HMI_DO(Sync := HMI.HMI_DO_Index<DO_Mapping.Do_End, HMI := HMI.HMI_DO_data, Local := GVL.Dout[HMI.HMI_DO_Index], strMode => HMI.HMI_DO_data.strMode, strStatus => HMI.HMI_DO_data.strStatus);
IF HMI_DO.ENO THEN
  DO_Name:=HMI.HMI_DO_Index;
  HMI.HMI_DO_Data.strName:=Burkert.Burkert_OSCAT_BASIC.REPLACE_ALL(str:=TO_STRING(DO_Name), src:='_' , rep:=' ' );
END_IF;

HMI_8098(Sync := HMI.HMI_8098_Index<s8098_Mapping.s8098_end, HMI := HMI.HMI_8098_Data, Local := PVL.s8098[HMI.HMI_8098_Index], strNamur => HMI.HMI_8098_Data.StrNamur107);
IF HMI_8098.ENO THEN
  S8098_Name:=HMI.HMI_8098_Index;
  HMI.HMI_8098_Data.strName:=Burkert.Burkert_OSCAT_BASIC.REPLACE_ALL(str:=TO_STRING(s8098_Name), src:='_' , rep:=' ' );
END_IF;

_Burkert_HMI_ME44AI_Sync187_OUT := Burkert.HMI_ME44AI_Sync(EN := HMI.HMI_ME44AI_Index<ME44AI_Mapping.ME44_AI_End, Local := Network.ME44_AI[HMI.HMI_ME44AI_Index], HMI := HMI.HMI_ME44AI_data, ENO => _Burkert_HMI_ME44AI_Sync187_ENO);
IF _Burkert_HMI_ME44AI_Sync187_ENO THEN
  ME44AI_Name:=HMI.HMI_ME44AI_Index;
  HMI.HMI_ME44AI_Data.strName:=Burkert.Burkert_OSCAT_BASIC.REPLACE_ALL(str:=TO_STRING(ME44AI_Name), src:='_' , rep:=' ' );
END_IF;
END_PROGRAM

PROGRAM VFD_Manager
  VAR
    VFD_101A_CTRL : Burkert.Eaton_DM1;
    VFD_101B_CTRL : Burkert.Eaton_DM1;
    VFD_102A_CTRL : Burkert.Eaton_DM1;
    VFD_102B_CTRL : Burkert.Eaton_DM1;
    VFD_102C_CTRL : Burkert.Eaton_DM1;
    VFD_102D_CTRL : Burkert.Eaton_DM1;
    VFD_102E_CTRL : Burkert.Eaton_DM1;
    VFD_102F_CTRL : Burkert.Eaton_DM1;
    VFD_102G_CTRL : Burkert.Eaton_DM1;
    VFD_102H_CTRL : Burkert.Eaton_DM1;
    VFD_201_CTRL : Burkert.Eaton_DM1;
    VFD_201B_CTRL : Burkert.Eaton_DM1;
    VFD_202_CTRL : Burkert.Eaton_DM1;
    VFD_202B_CTRL : Burkert.Eaton_DM1;
    VFD_203_CTRL : Burkert.Eaton_DM1;
  END_VAR

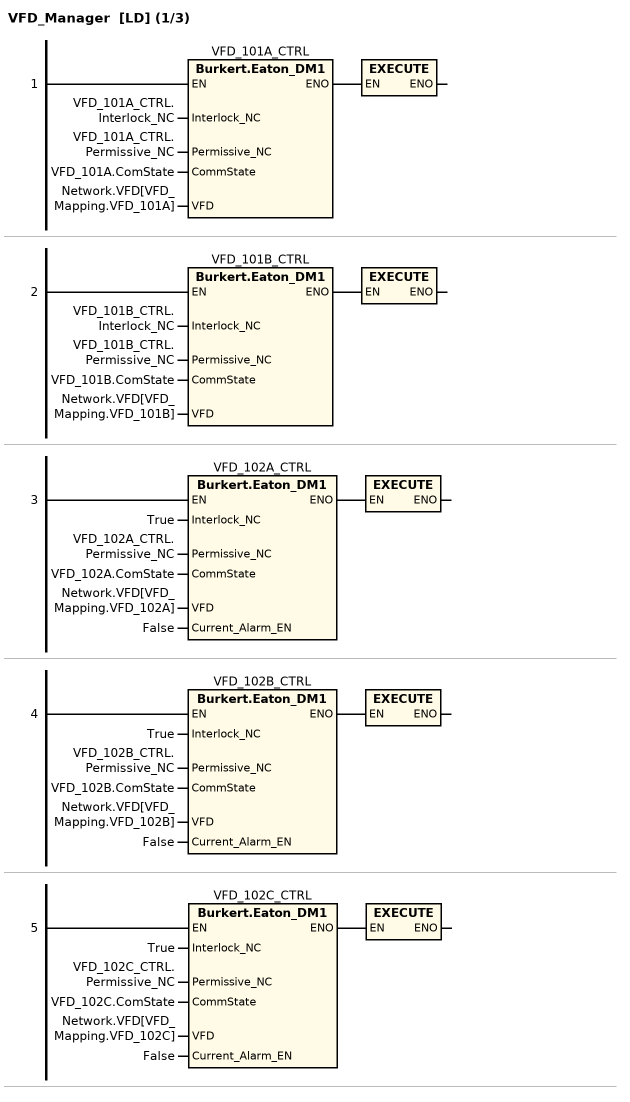
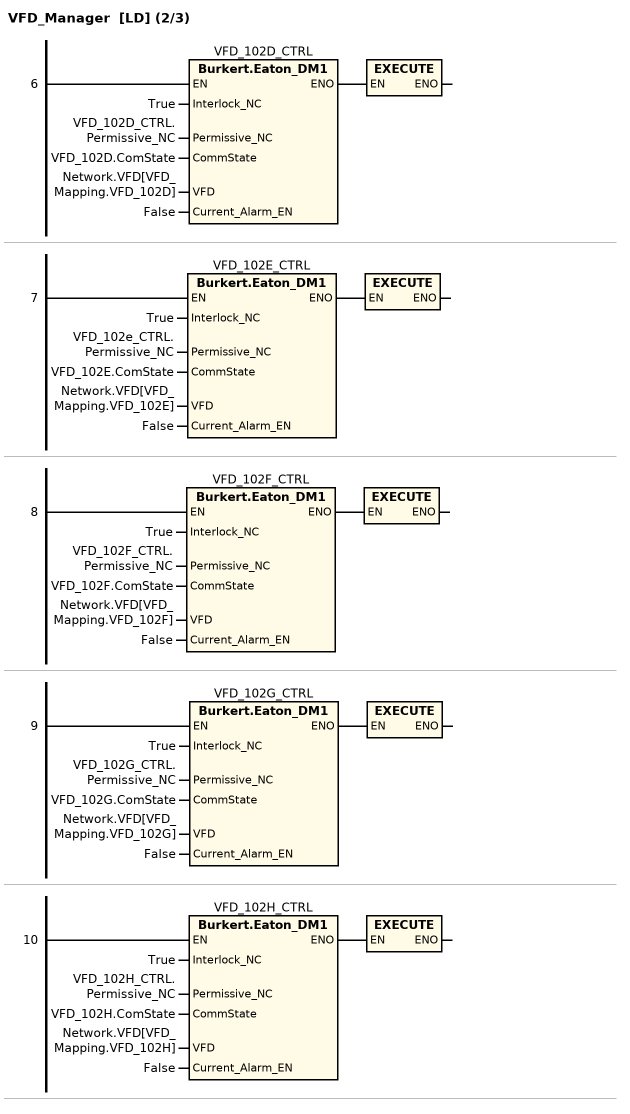
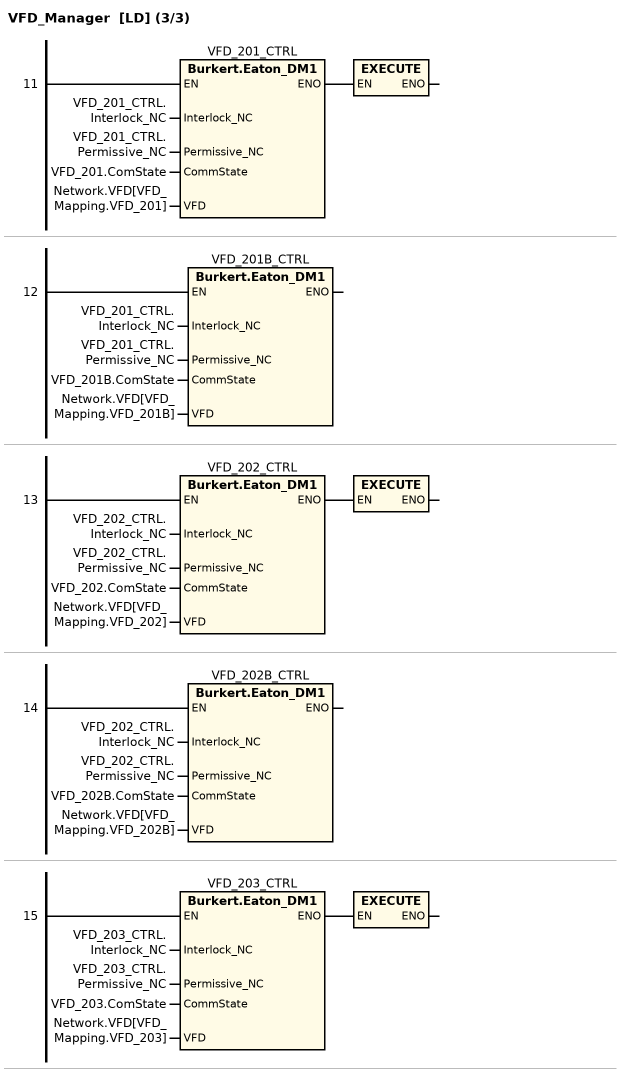
(* LD diagram, written out as Structured Text *)

VFD_101A_CTRL(Interlock_NC := VFD_101A_CTRL.Interlock_NC, Permissive_NC := VFD_101A_CTRL.Permissive_NC, CommState := VFD_101A.ComState, VFD := Network.VFD[VFD_Mapping.VFD_101A]);
IF VFD_101A_CTRL.ENO THEN
  VFD_101A_CTRL.Permissive_NC:= (GVL.s3363[s3363_mapping.ACV_101].Valve_Actual>5
  	) AND (
  	GVL.LS[LS_Mapping.LSLL_101].Status.eStatus=Burkert.DI_Status.Liquid_Detected AND
  	GVL.LS[Ls_mapping.LSHH_201].Status.eStatus=Burkert.DI_Status.No_Liquid_Detected);
  
  
  VFD_101A_CTRL.Interlock_NC:=TRUE;//(
  	//GVL.LS[LS_Mapping.LSLL_101].Status.eStatus=Burkert.DI_Status.Liquid_Detected AND
  	//GVL.LS[Ls_mapping.LSHH_201].Status.eStatus=Burkert.DI_Status.No_Liquid_Detected);
END_IF;

VFD_101B_CTRL(Interlock_NC := VFD_101B_CTRL.Interlock_NC, Permissive_NC := VFD_101B_CTRL.Permissive_NC, CommState := VFD_101B.ComState, VFD := Network.VFD[VFD_Mapping.VFD_101B]);
IF VFD_101B_CTRL.ENO THEN
  VFD_101B_CTRL.Permissive_NC:=(GVL.s3363[s3363_mapping.ACV_102].Valve_Actual>5 ) AND 
  	(GVL.LS[LS_Mapping.LSLL_101].Status.eStatus=Burkert.DI_Status.Liquid_Detected AND
  	GVL.LS[Ls_mapping.LSHH_201].Status.eStatus=Burkert.DI_Status.No_Liquid_Detected) ;
  	
  	VFD_101B_CTRL.Interlock_NC:=TRUE;//
  //(GVL.LS[LS_Mapping.LSLL_101].Status.eStatus=Burkert.DI_Status.Liquid_Detected AND GVL.LS[Ls_mapping.LSHH_201].Status.eStatus=Burkert.DI_Status.No_Liquid_Detected);
END_IF;

VFD_102A_CTRL(Interlock_NC := True, Permissive_NC := VFD_102A_CTRL.Permissive_NC, CommState := VFD_102A.ComState, VFD := Network.VFD[VFD_Mapping.VFD_102A], Current_Alarm_EN := False);
IF VFD_102A_CTRL.ENO THEN
  VFD_102A_CTRL.Permissive_NC:=(
  	NOT(PVL.AIT[AIT_Mapping.LT_101_P].Status.eStatus=Burkert.eSensor_Status.Low_Low_Alarm)
  	);
END_IF;

VFD_102B_CTRL(Interlock_NC := True, Permissive_NC := VFD_102B_CTRL.Permissive_NC, CommState := VFD_102B.ComState, VFD := Network.VFD[VFD_Mapping.VFD_102B], Current_Alarm_EN := False);
IF VFD_102B_CTRL.ENO THEN
  VFD_102B_CTRL.Permissive_NC:=(
  	NOT(PVL.AIT[AIT_Mapping.LT_101_P].Status.eStatus=Burkert.eSensor_Status.Low_Low_Alarm)
  	);
END_IF;

VFD_102C_CTRL(Interlock_NC := True, Permissive_NC := VFD_102C_CTRL.Permissive_NC, CommState := VFD_102C.ComState, VFD := Network.VFD[VFD_Mapping.VFD_102C], Current_Alarm_EN := False);
IF VFD_102C_CTRL.ENO THEN
  VFD_102C_CTRL.Permissive_NC:=(
  	NOT(PVL.AIT[AIT_Mapping.LT_101_P].Status.eStatus=Burkert.eSensor_Status.Low_Low_Alarm)
  	);
END_IF;

VFD_102D_CTRL(Interlock_NC := True, Permissive_NC := VFD_102D_CTRL.Permissive_NC, CommState := VFD_102D.ComState, VFD := Network.VFD[VFD_Mapping.VFD_102D], Current_Alarm_EN := False);
IF VFD_102D_CTRL.ENO THEN
  VFD_102D_CTRL.Permissive_NC:=(
  	NOT(PVL.AIT[AIT_Mapping.LT_101_P].Status.eStatus=Burkert.eSensor_Status.Low_Low_Alarm)
  	);
END_IF;

VFD_102E_CTRL(Interlock_NC := True, Permissive_NC := VFD_102e_CTRL.Permissive_NC, CommState := VFD_102E.ComState, VFD := Network.VFD[VFD_Mapping.VFD_102E], Current_Alarm_EN := False);
IF VFD_102E_CTRL.ENO THEN
  VFD_102E_CTRL.Permissive_NC:=(
  	NOT(PVL.AIT[AIT_Mapping.LT_201].Status.eStatus=Burkert.eSensor_Status.Low_Low_Alarm)
  	);
END_IF;

VFD_102F_CTRL(Interlock_NC := True, Permissive_NC := VFD_102F_CTRL.Permissive_NC, CommState := VFD_102F.ComState, VFD := Network.VFD[VFD_Mapping.VFD_102F], Current_Alarm_EN := False);
IF VFD_102F_CTRL.ENO THEN
  VFD_102F_CTRL.Permissive_NC:=(
  	NOT(PVL.AIT[AIT_Mapping.LT_201].Status.eStatus=Burkert.eSensor_Status.Low_Low_Alarm)
  	);
END_IF;

VFD_102G_CTRL(Interlock_NC := True, Permissive_NC := VFD_102G_CTRL.Permissive_NC, CommState := VFD_102G.ComState, VFD := Network.VFD[VFD_Mapping.VFD_102G], Current_Alarm_EN := False);
IF VFD_102G_CTRL.ENO THEN
  VFD_102G_CTRL.Permissive_NC:=(
  	NOT(PVL.AIT[AIT_Mapping.LT_201].Status.eStatus=Burkert.eSensor_Status.Low_Low_Alarm)
  	);
END_IF;

VFD_102H_CTRL(Interlock_NC := True, Permissive_NC := VFD_102H_CTRL.Permissive_NC, CommState := VFD_102H.ComState, VFD := Network.VFD[VFD_Mapping.VFD_102H], Current_Alarm_EN := False);
IF VFD_102H_CTRL.ENO THEN
  VFD_102H_CTRL.Permissive_NC:=(
  	NOT(PVL.AIT[AIT_Mapping.LT_201].Status.eStatus=Burkert.eSensor_Status.Low_Low_Alarm)
  	);
END_IF;

VFD_201_CTRL(Interlock_NC := VFD_201_CTRL.Interlock_NC, Permissive_NC := VFD_201_CTRL.Permissive_NC, CommState := VFD_201.ComState, VFD := Network.VFD[VFD_Mapping.VFD_201]);
IF VFD_201_CTRL.ENO THEN
  VFD_201_CTRL.Permissive_NC:=(GVL.s3363[s3363_mapping.ACV_201].Valve_Actual>10) AND 
  	(
  	(GVL.LS[LS_Mapping.LSHH_204].Status.eStatus=Burkert.DI_Status.No_Liquid_Detected OR GVL.LS[LS_Mapping.LSHH_204].Status.eStatus=Burkert.DI_Status.No_Liquid_Detected_Alarm) AND (GVL.LS[LS_mapping.LSLL_202].Status.eStatus=Burkert.DI_Status.Liquid_Detected)
  	);
  
  VFD_201_CTRL.Interlock_NC:=TRUE;//
  //((GVL.LS[LS_Mapping.LSHH_204].Status.eStatus=Burkert.DI_Status.No_Liquid_Detected OR GVL.LS[LS_Mapping.LSHH_204].Status.eStatus=Burkert.DI_Status.No_Liquid_Detected_Alarm) AND (GVL.LS[LS_mapping.LSLL_202].Status.eStatus=Burkert.DI_Status.Liquid_Detected));
END_IF;

VFD_201B_CTRL(Interlock_NC := VFD_201_CTRL.Interlock_NC, Permissive_NC := VFD_201_CTRL.Permissive_NC, CommState := VFD_201B.ComState, VFD := Network.VFD[VFD_Mapping.VFD_201B]);

VFD_202_CTRL(Interlock_NC := VFD_202_CTRL.Interlock_NC, Permissive_NC := VFD_202_CTRL.Permissive_NC, CommState := VFD_202.ComState, VFD := Network.VFD[VFD_Mapping.VFD_202]);
IF VFD_202_CTRL.ENO THEN
  VFD_202_CTRL.Permissive_NC:=(
  	(GVL.LS[LS_Mapping.LSLL_205].Status.eStatus=Burkert.DI_Status.Liquid_Detected) AND
  		(GVL.Filter_Path_Available OR 
  		(GVL.s3363[s3363_Mapping.ACV_203].Valve_Actual>5 AND GVL.s3363[s3363_Mapping.ACV_206].Valve_Actual>5)
  			)
  	);
  (*		
  		(GVL.s3363[s3363_Mapping.ACV_203].Valve_Actual>5 AND GVL.s3363[s3363_Mapping.ACV_206].Valve_Actual>5) OR
  		(	GVL.s3363[s3363_Mapping.ACV_207].Valve_Actual>5 OR
  			GVL.s3363[s3363_Mapping.ACV_208].Valve_Actual>5 OR
  			GVL.s3363[s3363_Mapping.ACV_213].Valve_Actual>5 OR
  			GVL.s3363[s3363_Mapping.ACV_214].Valve_Actual>5 OR
  			GVL.s3363[s3363_Mapping.ACV_219].Valve_Actual>5)
  	) AND	(
  		GVL.s3363[s3363_Mapping.ACV_224].Valve_Actual>5 OR
  		GVL.s3363[s3363_Mapping.ACV_225].Valve_Actual>5 OR
  		GVL.s3363[s3363_Mapping.ACV_226].Valve_Actual>5)	
  )	OR
  PVL.Z202_Config.Task.eTask=eZ202_Task.Drain_P202;
  *)
  
  
  
  VFD_202_CTRL.Interlock_NC:=TRUE;//(GVL.LS[LS_Mapping.LSLL_203].Status.eStatus=Burkert.DI_Status.Liquid_Detected);
END_IF;

VFD_202B_CTRL(Interlock_NC := VFD_202_CTRL.Interlock_NC, Permissive_NC := VFD_202_CTRL.Permissive_NC, CommState := VFD_202B.ComState, VFD := Network.VFD[VFD_Mapping.VFD_202B]);

VFD_203_CTRL(Interlock_NC := VFD_203_CTRL.Interlock_NC, Permissive_NC := VFD_203_CTRL.Permissive_NC, CommState := VFD_203.ComState, VFD := Network.VFD[VFD_Mapping.VFD_203]);
IF VFD_203_CTRL.ENO THEN
  VFD_203_CTRL.Permissive_NC:=(
  	(GVL.LS[LS_Mapping.LSLL_203].Status.eStatus=Burkert.DI_Status.Liquid_Detected) AND 
  	(GVL.s3363[s3363_Mapping.ACV_203].Valve_Actual>5 OR
  	(GVL.s3363[s3363_Mapping.ACV_206].Valve_Actual>6 AND GVL.Filter_Path_Available)
  	));// OR
  	//PVL.Z202_Config.Task.eTask=eZ202_Task.Drain_P203;
  	
  VFD_203_CTRL.Interlock_NC:=True;//(GVL.LS[LS_Mapping.LSLL_203].Status.eStatus=Burkert.DI_Status.Liquid_Detected);
END_IF;
END_PROGRAM

PROGRAM Stride_IO
  VAR
    Z201_RTD_Manager : Burkert.MB0_RTD;
    Z202_DO_Manager : Burkert.SIO_MB12CDR;
    tFIT : Burkert.cBase_FIT;
    tSensor : Burkert.cAnalog_Sensor;
  END_VAR

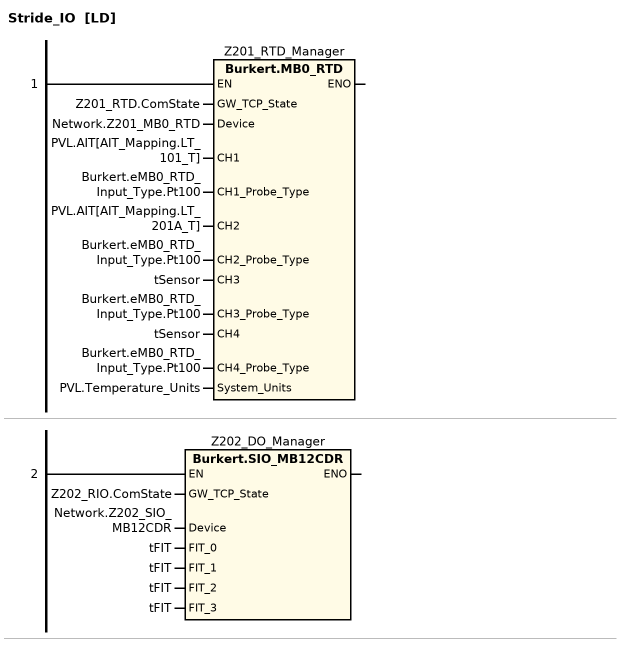
(* LD diagram, written out as Structured Text *)

Z201_RTD_Manager(GW_TCP_State := Z201_RTD.ComState, Device := Network.Z201_MB0_RTD, CH1 := PVL.AIT[AIT_Mapping.LT_101_T], CH1_Probe_Type := Burkert.eMB0_RTD_Input_Type.Pt100, CH2 := PVL.AIT[AIT_Mapping.LT_201A_T], CH2_Probe_Type := Burkert.eMB0_RTD_Input_Type.Pt100, CH3 := tSensor, CH3_Probe_Type := Burkert.eMB0_RTD_Input_Type.Pt100, CH4 := tSensor, CH4_Probe_Type := Burkert.eMB0_RTD_Input_Type.Pt100, System_Units := PVL.Temperature_Units);

Z202_DO_Manager(GW_TCP_State := Z202_RIO.ComState, Device := Network.Z202_SIO_MB12CDR, FIT_0 := tFIT, FIT_1 := tFIT, FIT_2 := tFIT, FIT_3 := tFIT);
END_PROGRAM

PROGRAM RCP_Manager
  VAR
    RecipeManCommands : RecipeManCommands;
    Save_Response : DWORD;
    Load_Response : DWORD;
    Storage_Response : BOOL;
    Load_Ton : ton;
    Save_Ton : Ton;
    Auto_Load_Ton : Ton;
    File_Save : BOOL;
    File_Save_Response : DWORD;
    R_Trig_0 : R_Trig;
    Save_R_trig : R_trig;
  END_VAR

            RecipeManCommands();
Storage_Response:=RecipeManCommands.SetStoragePath('RCP/');
//RecipeManCommands.GetRecipeNames(RecipeDefinitionName:='PersistentVariables',pStrings:=ADR(RCP_Names),iSize:=10,iStartIndex:=0);
Save_R_trig(CLK:=GVL.RCP_Save);
IF Save_R_trig.Q THEN 
	Save_Response:=16#FFFF; 
	PVL.RCP_Count:=PVL.RCP_Count+1;
END_IF;


IF GVL.RCP_Save THEN 
	//Save_Response:=16#FFFF;	
	Save_Response:=ReadAndSave();
	END_IF;
IF GVL.RCP_Load THEN	Load_Response:=LoadAndWrite(); END_IF;


Save_ton(In:=GVL.RCP_Save AND NOT(Save_Response=16#FFFF),PT:=T#2S);
IF Save_Ton.Q THEN GVL.RCP_Save:=FALSE; END_IF;




Load_ton(In:=GVL.RCP_Load,PT:=T#2S);
IF Load_Ton.Q THEN		
	GVL.RCP_Load :=FALSE;
	PVl.RCP_Loaded:=TRUE;
	END_IF;

Auto_Load_Ton(IN:=NOT(PVl.RCP_Loaded),PT:=T#10S);

IF Auto_load_Ton.Q THEN GVL.RCP_Load:=TRUE;	END_IF;
//IF GVL.Day_Seconds=30500 THEN GVL.RCP_Save:=TRUE; END_IF;
R_Trig_0(CLK:=GVL.RCP_Save);



//IF File_Save THEN 
//	File_Save_Response:=RecipeManCommands.SaveRecipe	(RecipeDefinitionName:='PersistentVariables',RecipeName:='Day_27');//,FileName:='BackUp_1.txtrecipe'); 
///END_IF;
          

METHOD ReadAndSave : DWORD
                  //ReadAndSave:=RecipeManCommands.ReadAndSaveRecipe(RecipeDefinitionName:='Vars',RecipeName:='BackUp');
//ReadAndSave:=RecipeManCommands.ReadRecipe	(RecipeDefinitionName:='PersistentVariables',RecipeName:='BackUp');
RecipeManCommands.CreateRecipe(RecipeDefinitionName:='Vars',RecipeName:='BackUp');
ReadAndSave:=RecipeManCommands.ReadAndSaveRecipeAs	(RecipeDefinitionName:='Vars',RecipeName:='BackUp',FileName:='BackUp.Vars.txtrecipe');

                
END_METHOD

METHOD LoadAndWrite : DWORD
                  //LoadAndWrite:=RecipeManCommands.LoadAndWriteRecipe(RecipeDefinitionName:='Recipes',RecipeName:='BackUp');

LoadAndWrite:=RecipeManCommands.LoadFromAndWriteRecipe(FileName:='BackUp.Vars.txtrecipe',RecipeDefinitionName:='Vars',RecipeName:='BackUp');
                
END_METHOD
END_PROGRAM

PROGRAM LS_Manager
  VAR
    LSHH_201_CTRL : Burkert.LS_UDFB;
    LSLL_202_CTRL : Burkert.LS_UDFB;
    LSLL_101_CTRL : Burkert.LS_UDFB;
    LSHH_206_CTRL : Burkert.LS_UDFB;
    LSLL_210_CTRL : Burkert.LS_UDFB;
    LSHH_208_CTRL : Burkert.LS_UDFB;
    LSLL_212_CTRL : Burkert.LS_UDFB;
    LSHH_209_CTRL : Burkert.LS_UDFB;
    LSLL_213_CTRL : Burkert.LS_UDFB;
    LSHH_207_CTRL : Burkert.LS_UDFB;
    LSLL_211_CTRL : Burkert.LS_UDFB;
    LSHH_204_CTRL : Burkert.LS_UDFB;
    LSLL_205_CTRL : Burkert.LS_UDFB;
    LSLL_203_CTRL : Burkert.LS_UDFB;
  END_VAR

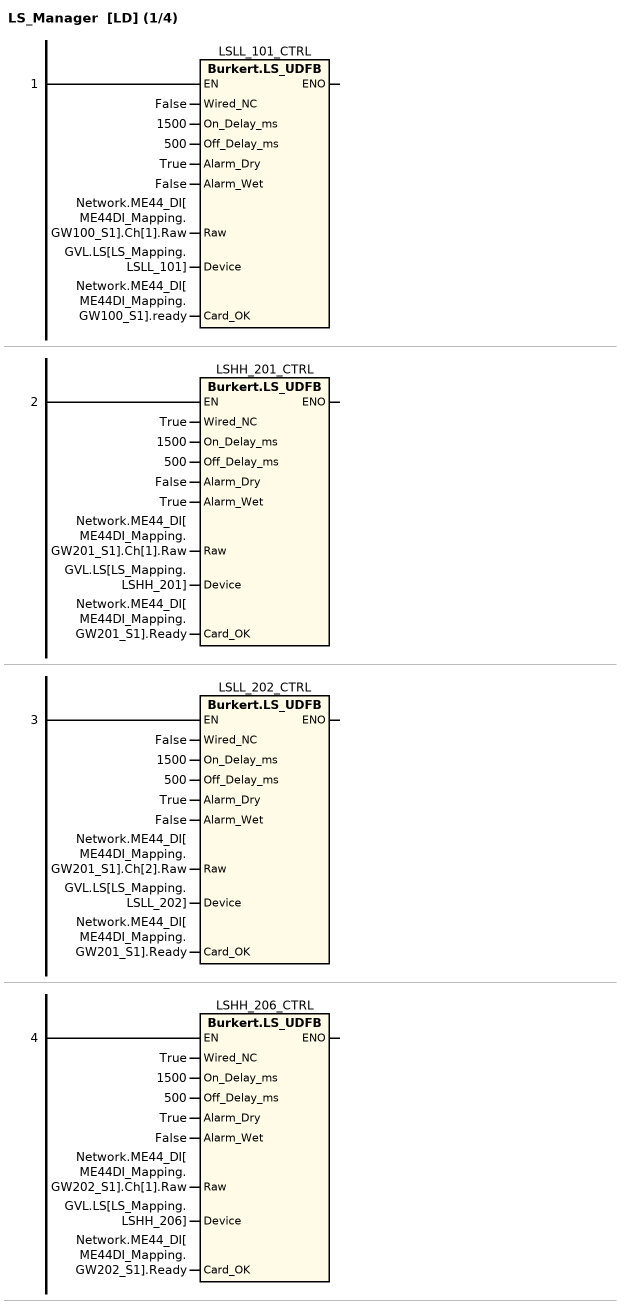
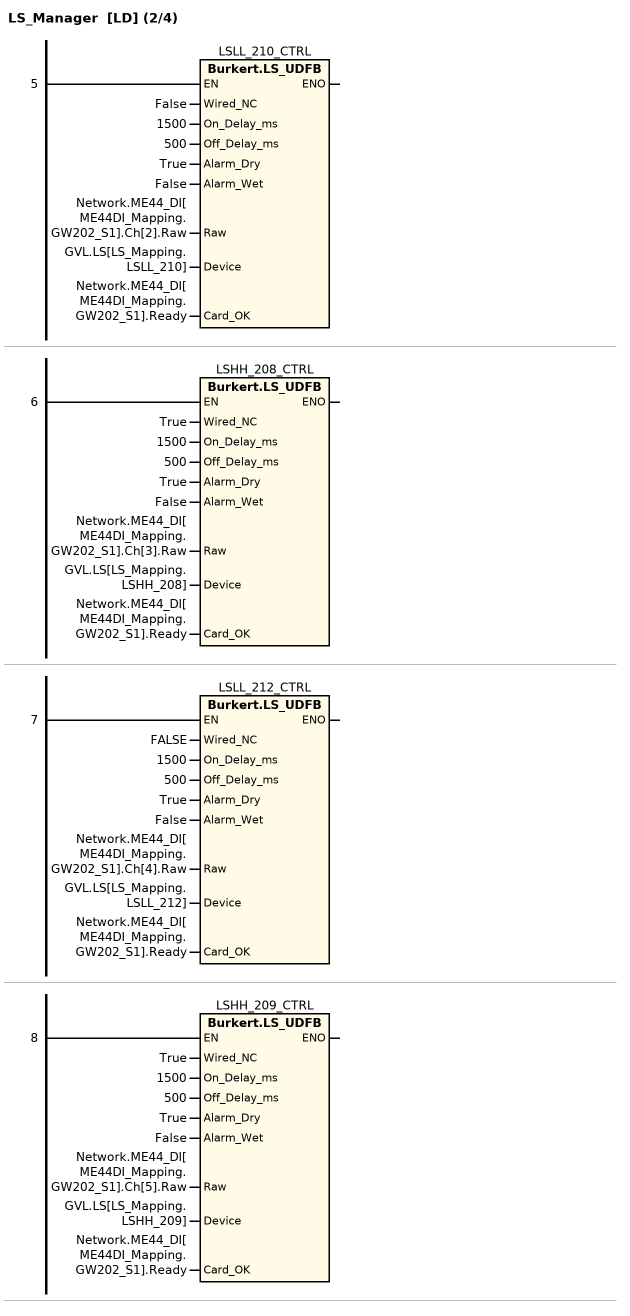
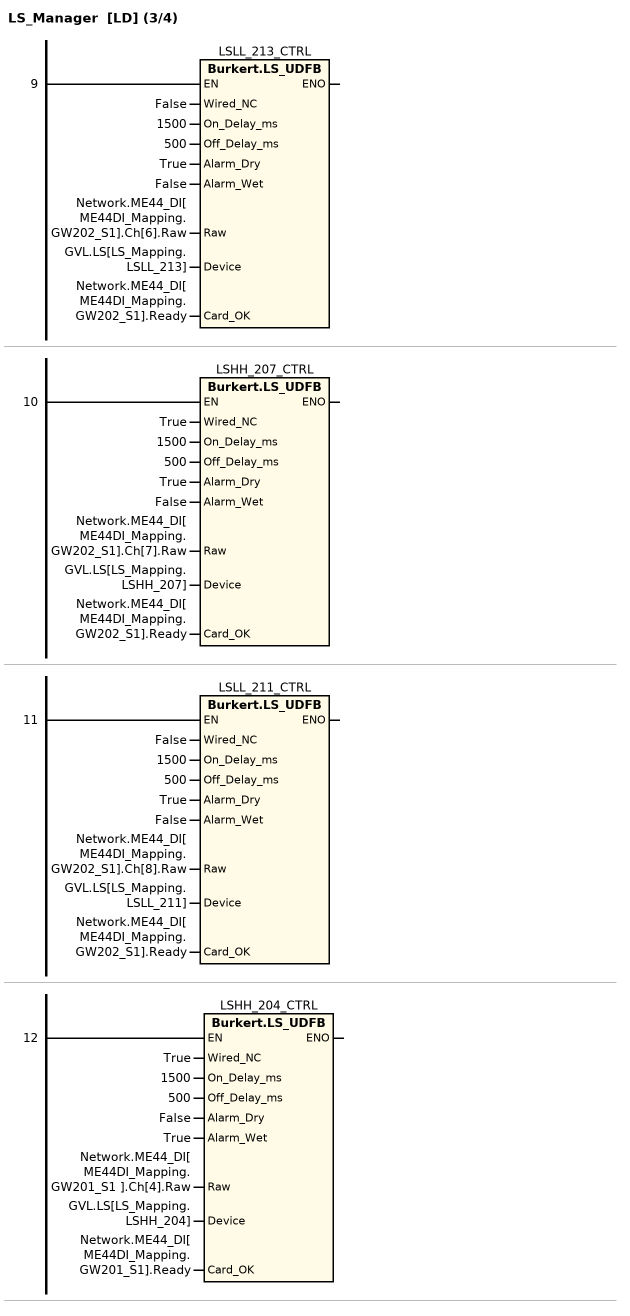
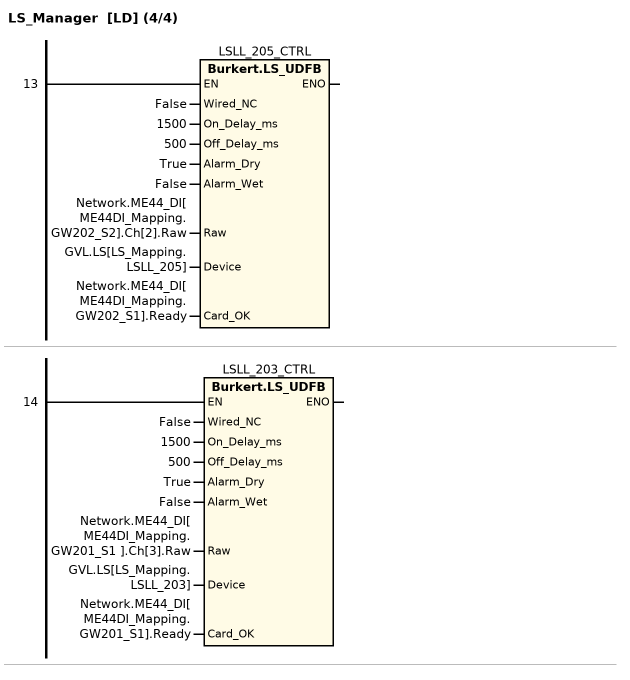
(* LD diagram, written out as Structured Text *)

LSLL_101_CTRL(Wired_NC := False, On_Delay_ms := 1500, Off_Delay_ms := 500, Alarm_Dry := True, Alarm_Wet := False, Raw := Network.ME44_DI[ME44DI_Mapping.GW100_S1].Ch[1].Raw, Device := GVL.LS[LS_Mapping.LSLL_101], Card_OK := Network.ME44_DI[ME44DI_Mapping.GW100_S1].ready);

LSHH_201_CTRL(Wired_NC := True, On_Delay_ms := 1500, Off_Delay_ms := 500, Alarm_Dry := False, Alarm_Wet := True, Raw := Network.ME44_DI[ME44DI_Mapping.GW201_S1].Ch[1].Raw, Device := GVL.LS[LS_Mapping.LSHH_201], Card_OK := Network.ME44_DI[ME44DI_Mapping.GW201_S1].Ready);

LSLL_202_CTRL(Wired_NC := False, On_Delay_ms := 1500, Off_Delay_ms := 500, Alarm_Dry := True, Alarm_Wet := False, Raw := Network.ME44_DI[ME44DI_Mapping.GW201_S1].Ch[2].Raw, Device := GVL.LS[LS_Mapping.LSLL_202], Card_OK := Network.ME44_DI[ME44DI_Mapping.GW201_S1].Ready);

LSHH_206_CTRL(Wired_NC := True, On_Delay_ms := 1500, Off_Delay_ms := 500, Alarm_Dry := True, Alarm_Wet := False, Raw := Network.ME44_DI[ME44DI_Mapping.GW202_S1].Ch[1].Raw, Device := GVL.LS[LS_Mapping.LSHH_206], Card_OK := Network.ME44_DI[ME44DI_Mapping.GW202_S1].Ready);

LSLL_210_CTRL(Wired_NC := False, On_Delay_ms := 1500, Off_Delay_ms := 500, Alarm_Dry := True, Alarm_Wet := False, Raw := Network.ME44_DI[ME44DI_Mapping.GW202_S1].Ch[2].Raw, Device := GVL.LS[LS_Mapping.LSLL_210], Card_OK := Network.ME44_DI[ME44DI_Mapping.GW202_S1].Ready);

LSHH_208_CTRL(Wired_NC := True, On_Delay_ms := 1500, Off_Delay_ms := 500, Alarm_Dry := True, Alarm_Wet := False, Raw := Network.ME44_DI[ME44DI_Mapping.GW202_S1].Ch[3].Raw, Device := GVL.LS[LS_Mapping.LSHH_208], Card_OK := Network.ME44_DI[ME44DI_Mapping.GW202_S1].Ready);

LSLL_212_CTRL(Wired_NC := FALSE, On_Delay_ms := 1500, Off_Delay_ms := 500, Alarm_Dry := True, Alarm_Wet := False, Raw := Network.ME44_DI[ME44DI_Mapping.GW202_S1].Ch[4].Raw, Device := GVL.LS[LS_Mapping.LSLL_212], Card_OK := Network.ME44_DI[ME44DI_Mapping.GW202_S1].Ready);

LSHH_209_CTRL(Wired_NC := True, On_Delay_ms := 1500, Off_Delay_ms := 500, Alarm_Dry := True, Alarm_Wet := False, Raw := Network.ME44_DI[ME44DI_Mapping.GW202_S1].Ch[5].Raw, Device := GVL.LS[LS_Mapping.LSHH_209], Card_OK := Network.ME44_DI[ME44DI_Mapping.GW202_S1].Ready);

LSLL_213_CTRL(Wired_NC := False, On_Delay_ms := 1500, Off_Delay_ms := 500, Alarm_Dry := True, Alarm_Wet := False, Raw := Network.ME44_DI[ME44DI_Mapping.GW202_S1].Ch[6].Raw, Device := GVL.LS[LS_Mapping.LSLL_213], Card_OK := Network.ME44_DI[ME44DI_Mapping.GW202_S1].Ready);

LSHH_207_CTRL(Wired_NC := True, On_Delay_ms := 1500, Off_Delay_ms := 500, Alarm_Dry := True, Alarm_Wet := False, Raw := Network.ME44_DI[ME44DI_Mapping.GW202_S1].Ch[7].Raw, Device := GVL.LS[LS_Mapping.LSHH_207], Card_OK := Network.ME44_DI[ME44DI_Mapping.GW202_S1].Ready);

LSLL_211_CTRL(Wired_NC := False, On_Delay_ms := 1500, Off_Delay_ms := 500, Alarm_Dry := True, Alarm_Wet := False, Raw := Network.ME44_DI[ME44DI_Mapping.GW202_S1].Ch[8].Raw, Device := GVL.LS[LS_Mapping.LSLL_211], Card_OK := Network.ME44_DI[ME44DI_Mapping.GW202_S1].Ready);

LSHH_204_CTRL(Wired_NC := True, On_Delay_ms := 1500, Off_Delay_ms := 500, Alarm_Dry := False, Alarm_Wet := True, Raw := Network.ME44_DI[ME44DI_Mapping.GW201_S1 ].Ch[4].Raw, Device := GVL.LS[LS_Mapping.LSHH_204], Card_OK := Network.ME44_DI[ME44DI_Mapping.GW201_S1].Ready);

LSLL_205_CTRL(Wired_NC := False, On_Delay_ms := 1500, Off_Delay_ms := 500, Alarm_Dry := True, Alarm_Wet := False, Raw := Network.ME44_DI[ME44DI_Mapping.GW202_S2].Ch[2].Raw, Device := GVL.LS[LS_Mapping.LSLL_205], Card_OK := Network.ME44_DI[ME44DI_Mapping.GW202_S1].Ready);

LSLL_203_CTRL(Wired_NC := False, On_Delay_ms := 1500, Off_Delay_ms := 500, Alarm_Dry := True, Alarm_Wet := False, Raw := Network.ME44_DI[ME44DI_Mapping.GW201_S1 ].Ch[3].Raw, Device := GVL.LS[LS_Mapping.LSLL_203], Card_OK := Network.ME44_DI[ME44DI_Mapping.GW201_S1].Ready);
(* --- network --- *)
END_PROGRAM

PROGRAM Level_3_CTRL

            Z100_Manager();
Z201_Manager();
Z202_Manager();
Filter_manager();





          
END_PROGRAM

PROGRAM Z100_Manager
  VAR
    Local_Status : eZ100_Status;
    tStatus : eZ100_Status;
    Local_Task : eZ100_Task;
    FT101_Ave : REAL;
    FT101_Hav : REAL;
    FT101_Ave_Index : INT;
    FT101_Array_Size : UINT;
  END_VAR
  VAR  (* added by the conversion: wires and edge detectors of the diagram *)
    _OR2_OUT : BOOL;
  END_VAR

            
PVL.Z100_Config.StrMode:=Burkert.Burkert_OSCAT_BASIC.REPLACE_ALL(str:=TO_STRING(PVL.Z100_Config.Mode.eMode) , src:='_' , rep:=' ' );
PVL.Z100_Config.StrStatus:=Burkert.Burkert_OSCAT_BASIC.REPLACE_ALL(str:=TO_STRING(PVL.Z100_Config.Status.eStatus) , src:='_' , rep:=' ' );
PVl.Z100_Config.StrTask:=Burkert.Burkert_OSCAT_BASIC.REPLACE_ALL(str:=TO_STRING(PVL.Z100_Config.Task.eTask) , src:='_' , rep:=' ' );
PVL.Z100_Config.Mode.eMode:=Burkert.eHOA_Modes.Manual;
Alarms();

CASE	PVL.Z100_Config.Task.eTask OF
	eZ100_task.Off: Task_OFF();
	eZ100_Task.Continuous_Level:Task_Level();
	eZ100_Task.Continuous_Flow_Intake:
	eZ100_Task.Continuous_Flow_Discharge: TASK_Flow_Discharge();
	eZ100_task.Continuous_UV:Continuous_UV();
	eZ100_Task.Batch_Level:
	eZ100_Task.Batch:
	eZ100_Task.Drain:Task_Drain();
END_CASE

PID_Manager();
ACV_Manager();

PVl.Duplex[Duplex_mapping.Z100].Run_Pct:=MAX(
	PVL.PID[pid_mapping.Z100_Flow].CV,
	PVl.PID[PID_Mapping.Z100_Level].CV,
	PVl.PID[PID_mapping.Z100_Pressure].CV);
PVl.Duplex[Duplex_Mapping.Z100].Run_Request:=PVl.Duplex[Duplex_mapping.Z100].Run_Pct>5;

pvl.Z100_Config.UV_Rate.Target:=SEL(
	PVL.Z100_Config.uvDSP>0,
	0,
	((0.06 * PVL.Z202_Config.Pond_Area_m2 * PVL.AIT[ait_Mapping.UV_001].EU) / PVL.Z100_Config.uvDSP));	
FT101_Array_Size:=SIZEOF(GVl.FT101_Ave);
IF GVL.CLK_500ms THEN
	IF FT101_Ave_Index<50 AND PVL.s8098[s8098_Mapping.FT_101].PDO.VolumeFlow.EU> 0 THEN	
		GVl.FT101_Ave[FT101_Ave_Index]:=PVL.s8098[s8098_Mapping.FT_101].PDO.VolumeFlow.EU;
		FT101_Ave_Index:=FT101_Ave_Index+1;
	ELSE
		Burkert.MEM.MemMove(pSource:= ADR(GVl.FT101_Ave[1]), pDestination:=ADR(GVl.FT101_Ave[0]) , uiNumberOfBytes:=(SIZEOF(GVl.FT101_Ave)-4) );
		GVl.FT101_Ave[49]:=PVL.s8098[s8098_Mapping.FT_101].PDO.VolumeFlow.EU;
	END_IF;

	IF FT101_Ave_Index>0 THEN
		FT101_Ave:=Burkert.Burkert_OSCAT_BASIC.ARRAY_AVG (	pt:=ADR(GVl.FT101_Ave),	size:=SIZEOF(GVl.FT101_Ave));
		FT101_Hav:=Burkert.Burkert_OSCAT_BASIC.ARRAY_HAV (	pt:=ADR(GVl.FT101_Ave[0]),size:=TO_UINT(FT101_Ave_Index*4));
	END_IF;
	
END_IF;

IF FT101_Ave=0  THEN 	FT101_Ave_Index:=0; END_IF;
PVl.PID[pid_mapping.Z100_Flow].Actual:=PVL.s8098[s8098_Mapping.FT_101].PDO.VolumeFlow.EU;;//FT101_AVE;
          

ACTION Evaluate_Batch_Level:
                tStatus:=Local_status;

//IF NOT(pvl.AIT[AIT_Mapping.LT_01A].Ready) 	THEN tStatus:=eZ100_Status.LT01A_Not_Ready; END_IF;
//IF NOT(pvl.AIT[AIT_Mapping.LT_01B].Ready) 	THEN tStatus:=eZ100_Status.LT01B_Not_Ready; END_IF;
IF NOT(pvl.AIT[AIT_Mapping.LT_101_P].Ready) 	THEN tStatus:=eZ100_Status.LT101_Not_Ready; END_IF;
IF PVL.AIT[AIT_Mapping.LT_101_P].Status.eStatus=Burkert.eSensor_Status.HiHi_Alarm THEN	tStatus:=eZ100_Status.EP101_LT101_High_High_Level_Alarm; END_IF;

//IF NOT(PVL.AIT[AIT_Mapping.FT_01].Ready) 	THEN tStatus:=eZ100_Status.FT01_Not_Ready; END_IF;
IF GVL.LS[LS_Mapping.LSLL_101].Status.eStatus=Burkert.DI_Status.No_Liquid_Detected_Alarm THEN	tStatus:=eZ100_Status.LSLL101_Pump_Intakes_Dry; END_IF;
IF NOT(Network.VFD[VFD_Mapping.VFD_101A].Ready) AND NOT(Network.VFD[VFD_Mapping.VFD_101B].Ready) THEN
	IF NOT(Network.VFD[VFD_Mapping.VFD_101A].Ready)	 	THEN	tStatus:=eZ100_Status.Pump_101A_Not_Ready; END_IF;
	IF NOT(Network.VFD[VFD_Mapping.VFD_101B].Ready) 	THEN	tStatus:=eZ100_Status.Pump_101B_Not_Ready; END_IF;
END_IF;
IF NOT(GVL.s3363[s3363_Mapping.ACV_101].Ready) AND NOT(GVL.s3363[s3363_Mapping.ACV_102].Ready) THEN
	IF NOT(GVL.s3363[s3363_Mapping.ACV_101].Ready) 		THEN	tStatus:=ez100_Status.ACV101_Not_Ready;END_IF;
	IF NOT(GVL.s3363[s3363_Mapping.ACV_102].Ready) 		THEN	tStatus:=ez100_Status.ACV102_Not_Ready;END_IF;
END_IF;
IF NOT(PVL.s8312[s8312_mapping.PT_101].Ready) 		THEN 	tStatus:=eZ100_Status.PT101_Not_Ready; END_IF;
IF NOT(PVL.s8098[s8098_Mapping.FT_101].Ready)		THEN	tStatus:=eZ100_Status.FT101_Not_Ready; END_IF;


IF GVL.LS[LS_Mapping.LSHH_201].Status.eStatus= Burkert.DI_Status.Liquid_Detected_Alarm THEN tStatus:=eZ100_Status.EP101_LSHH201_High_High_Level_Alarm; END_IF;
//IF PVL.AIT[AIT_Mapping.LT_01A].Status.eStatus=Burkert.eSensor_Status.Low_Low_Alarm THEN tStatus:=eZ100_Status.LT01A_Low_Low_Level_Alarm; END_IF;
//IF PVL.AIT[AIT_Mapping.LT_01B].Status.eStatus=Burkert.eSensor_Status.Low_Low_Alarm THEN tStatus:=eZ100_Status.LT01B_Low_Low_Level_Alarm; END_IF;
IF PVL.s8312[s8312_Mapping.PT_101].Status.eStatus=Burkert.eSensor_Status.Low_Low_Alarm THEN tStatus:=eZ100_Status.PT101_Low_Low_Pressure_Alarm; END_IF;
IF PVL.s8312[s8312_Mapping.PT_101].Status.eStatus=Burkert.eSensor_Status.HiHi_Alarm THEN tStatus:=eZ100_Status.PT101_High_High_Pressure_Alarm; END_IF;

IF PVl.Duplex[Duplex_mapping.Z100].Mode.eMode=Burkert.eDuplex_Mode.Disabled THEN	tStatus:=eZ100_Status.Pump_Duplex_Disabled; END_IF;

IF NOT(PVL.s8098[s8098_mapping.FT_101].Ready)	THEN	tStatus:=eZ100_Status.FT01_Not_Ready; END_IF;
IF PVl.s8098[s8098_mapping.FT_101].PDO.VolumeFlow.Status.eStatus=Burkert.eSensor_Status.Low_Low_Alarm THEN tStatus:=eZ100_Status.FT101_Low_Low_Flow_Alarm; END_IF;

PVl.Z100_Config.Status.eStatus:=tStatus;




              
END_ACTION

ACTION PID_Manager:
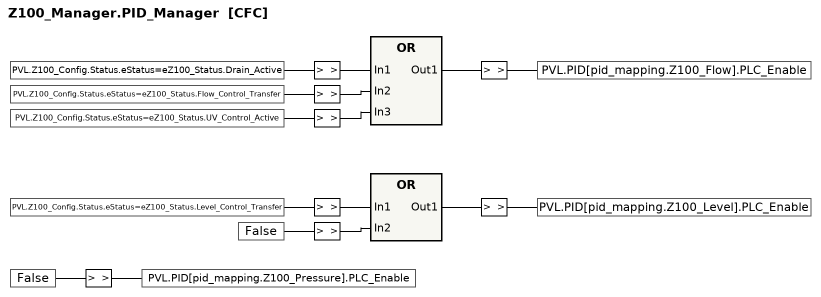
(* CFC diagram, written out as Structured Text *)
PVL.PID[pid_mapping.Z100_Flow].PLC_Enable := _OR2_OUT;
PVL.PID[pid_mapping.Z100_Level].PLC_Enable := (PVL.Z100_Config.Status.eStatus=eZ100_Status.Level_Control_Transfer) OR False;
PVL.PID[pid_mapping.Z100_Pressure].PLC_Enable := False;
_OR2_OUT := (PVL.Z100_Config.Status.eStatus=eZ100_Status.Drain_Active) OR (PVL.Z100_Config.Status.eStatus=eZ100_Status.Flow_Control_Transfer) OR (PVL.Z100_Config.Status.eStatus=eZ100_Status.UV_Control_Active);
END_ACTION

ACTION Task_Drain:
                IF PVL.Z100_Config.Task.eTask<> Local_Task THEN
	Local_Task:=PVL.Z100_Config.Task.eTask;
	PVL.Z100_Config.READY:=TRUE;
END_IF;






local_status:=eZ100_Status.Drain_Active;
PVL.PID[PID_Mapping.Z100_Flow].PLC_Target:=PVL.Z100_Config.Drain_Rate.Target;
Burkert.Alarm_Window_Convert(window:=PVL.Z100_Config.Drain_Rate,Config:=PVL.s8098[s8098_Mapping.FT_101].PDO.VolumeFlow.Alarm_Config);
Evaluate_Drain();


CASE PVL.Z100_Config.Status.eStatus OF
	//eZ100_Status.EP101_High_High_Level_Alarm: Local_Status:=eZ100_Status.EP101_High_High_Level_Alarm;
	//eZ100_Status.LT01A_Low_Low_Level_Alarm:			Local_Status:=eZ100_Status.LT01A_Low_Low_Level_Alarm;
	//eZ100_Status.LT01B_Low_Low_Level_Alarm:			Local_Status:=eZ100_Status.LT01B_Low_Low_Level_Alarm;
	eZ100_Status.PT101_High_High_Pressure_Alarm:	Local_Status:=eZ100_Status.PT101_High_High_Pressure_Alarm;PVL.Z100_Config.READY:=FALSE;
	eZ100_Status.PT101_Low_Low_Pressure_Alarm:		Local_Status:=eZ100_Status.PT101_Low_Low_Pressure_Alarm;PVL.Z100_Config.READY:=FALSE;
	eZ100_Status.LSLL101_Pump_Intakes_Dry:					Local_Status:=PVL.Z100_Config.Status.eStatus;PVL.Z100_Config.READY:=FALSE;
	eZ100_Status.Drain_Complete:					Local_Status:=PVL.Z100_Config.Status.eStatus;	PVL.Z100_Config.READY:=TRUE;
	eZ100_Status.Drain_Active:PVL.Z100_Config.READY:=TRUE;

END_CASE
              
END_ACTION

ACTION Evaluate_ALL:
                tStatus:=Local_status;

//IF NOT(pvl.AIT[AIT_Mapping.LT_01A].Ready) 	THEN tStatus:=eZ100_Status.LT01A_Not_Ready; END_IF;
//IF NOT(pvl.AIT[AIT_Mapping.LT_01B].Ready) 	THEN tStatus:=eZ100_Status.LT01B_Not_Ready; END_IF;
IF NOT(pvl.AIT[AIT_Mapping.LT_101_P].Ready) 	THEN tStatus:=eZ100_Status.LT101_Not_Ready; END_IF;
IF PVL.AIT[AIT_Mapping.LT_101_P].Status.eStatus=Burkert.eSensor_Status.HiHi_Alarm THEN	tStatus:=eZ100_Status.EP101_LT101_High_High_Level_Alarm; END_IF;

IF NOT(PVL.AIT[AIT_Mapping.FT_01].Ready) 	THEN tStatus:=eZ100_Status.FT01_Not_Ready; END_IF;
IF GVL.LS[LS_Mapping.LSLL_101].Status.eStatus=Burkert.DI_Status.No_Liquid_Detected_Alarm THEN	tStatus:=eZ100_Status.LSLL101_Pump_Intakes_Dry; END_IF;
IF NOT(Network.VFD[VFD_Mapping.VFD_101A].Ready)	 	THEN	tStatus:=eZ100_Status.Pump_101A_Not_Ready; END_IF;
IF NOT(Network.VFD[VFD_Mapping.VFD_101B].Ready) 	THEN	tStatus:=eZ100_Status.Pump_101B_Not_Ready; END_IF;
IF NOT(GVL.s3363[s3363_Mapping.ACV_101].Ready) 		THEN	tStatus:=ez100_Status.ACV101_Not_Ready;END_IF;
IF NOT(GVL.s3363[s3363_Mapping.ACV_102].Ready) 		THEN	tStatus:=ez100_Status.ACV102_Not_Ready;END_IF;
IF NOT(PVL.s8312[s8312_mapping.PT_101].Ready) 		THEN 	tStatus:=eZ100_Status.PT101_Not_Ready; END_IF;
IF NOT(PVL.s8098[s8098_Mapping.FT_101].Ready)		THEN	tStatus:=eZ100_Status.FT101_Not_Ready; END_IF;


IF GVL.LS[LS_Mapping.LSHH_201].Status.eStatus= Burkert.DI_Status.Liquid_Detected_Alarm THEN tStatus:=eZ100_Status.EP101_LSHH201_High_High_Level_Alarm; END_IF;
//IF PVL.AIT[AIT_Mapping.LT_01A].Status.eStatus=Burkert.eSensor_Status.Low_Low_Alarm THEN tStatus:=eZ100_Status.LT01A_Low_Low_Level_Alarm; END_IF;
//IF PVL.AIT[AIT_Mapping.LT_01B].Status.eStatus=Burkert.eSensor_Status.Low_Low_Alarm THEN tStatus:=eZ100_Status.LT01B_Low_Low_Level_Alarm; END_IF;
IF PVL.s8312[s8312_Mapping.PT_101].Status.eStatus=Burkert.eSensor_Status.Low_Low_Alarm THEN tStatus:=eZ100_Status.PT101_Low_Low_Pressure_Alarm; END_IF;
IF PVL.s8312[s8312_Mapping.PT_101].Status.eStatus=Burkert.eSensor_Status.HiHi_Alarm THEN tStatus:=eZ100_Status.PT101_High_High_Pressure_Alarm; END_IF;
IF PVl.Duplex[Duplex_mapping.Z100].Mode.eMode=Burkert.eDuplex_Mode.Disabled THEN	tStatus:=eZ100_Status.Pump_Duplex_Disabled; END_IF;

IF NOT(PVL.s8098[s8098_mapping.FT_101].Ready)	THEN	tStatus:=eZ100_Status.FT01_Not_Ready; END_IF;
IF PVl.s8098[s8098_mapping.FT_101].PDO.VolumeFlow.Status.eStatus=Burkert.eSensor_Status.Low_Low_Alarm THEN tStatus:=eZ100_Status.FT101_Low_Low_Flow_Alarm; END_IF;




PVl.Z100_Config.Status.eStatus:=tStatus;




              
END_ACTION

ACTION Continuous_UV:
                IF PVL.Z100_Config.Task.eTask<> Local_Task THEN
	Local_Task:=PVL.Z100_Config.Task.eTask;
	local_status:=eZ100_Status.UV_Control_Active;
END_IF;








PVL.PID[PID_Mapping.Z100_Flow].PLC_Target:=LIMIT(PVl.Z100_Config.UvLowerLimit, pvl.Z100_Config.UV_Rate.Target,PVl.Z100_Config.UvUpperLimit);
	

//Burkert.Alarm_Window_Convert(window:=PVL.Z100_Config.Target_Flow,Config:=PVL.s8098[s8098_Mapping.FT_101].PDO.VolumeFlow.Alarm_Config);
Evaluate_Continuous_UV();


CASE PVL.Z100_Config.Status.eStatus OF
	eZ100_Status.EP101_LSHH201_High_High_Level_Alarm: Local_Status:=eZ100_Status.EP101_LSHH201_High_High_Level_Alarm;
	//eZ100_Status.LT01A_Low_Low_Level_Alarm:			Local_Status:=eZ100_Status.LT01A_Low_Low_Level_Alarm;
	//eZ100_Status.LT01B_Low_Low_Level_Alarm:			Local_Status:=eZ100_Status.LT01B_Low_Low_Level_Alarm;
	eZ100_Status.PT101_High_High_Pressure_Alarm:	Local_Status:=eZ100_Status.PT101_High_High_Pressure_Alarm;
	//eZ100_Status.PT101_Low_Low_Pressure_Alarm:		Local_Status:=eZ100_Status.PT101_Low_Low_Pressure_Alarm;
	eZ100_Status.LSLL101_Pump_Intakes_Dry:					Local_Status:=eZ100_Status.LSLL101_Pump_Intakes_Dry;

END_CASE;

              
END_ACTION

ACTION Evaluate_Continuous_UV:
                tStatus:=Local_status;

//IF NOT(pvl.AIT[AIT_Mapping.LT_01A].Ready) 	THEN tStatus:=eZ100_Status.LT01A_Not_Ready; END_IF;
//IF NOT(pvl.AIT[AIT_Mapping.LT_01B].Ready) 	THEN tStatus:=eZ100_Status.LT01B_Not_Ready; END_IF;
IF NOT(pvl.AIT[AIT_Mapping.LT_101_P].Ready) 	THEN tStatus:=eZ100_Status.LT101_Not_Ready; END_IF;
IF PVL.AIT[AIT_Mapping.LT_101_P].Status.eStatus=Burkert.eSensor_Status.HiHi_Alarm THEN	tStatus:=eZ100_Status.EP101_LT101_High_High_Level_Alarm; END_IF;

//IF NOT(PVL.AIT[AIT_Mapping.FT_01].Ready) 	THEN tStatus:=eZ100_Status.FT01_Not_Ready; END_IF;
//IF NOT(PVL.AIT[Ait_mapping.UV_001].Ready)	THEN	tStatus:=ez100_status.UV_Sensor_Not_Ready;	END_IF;
//IF PVL.AIT[Ait_mapping.UV_001].EU=0	THEN	tStatus:=ez100_status.UV_Sensor_Error;	END_IF;
IF GVL.LS[LS_Mapping.LSLL_101].Status.eStatus=Burkert.DI_Status.No_Liquid_Detected_Alarm THEN	tStatus:=eZ100_Status.LSLL101_Pump_Intakes_Dry; END_IF;

IF NOT(Network.VFD[VFD_Mapping.VFD_101A].Ready) AND NOT(Network.VFD[VFD_Mapping.VFD_101B].Ready) THEN
	IF NOT(Network.VFD[VFD_Mapping.VFD_101A].Ready)	 	THEN	tStatus:=eZ100_Status.Pump_101A_Not_Ready; END_IF;
	IF NOT(Network.VFD[VFD_Mapping.VFD_101B].Ready) 	THEN	tStatus:=eZ100_Status.Pump_101B_Not_Ready; END_IF;
END_IF;
IF NOT(GVL.s3363[s3363_Mapping.ACV_101].Ready) AND NOT(GVL.s3363[s3363_Mapping.ACV_102].Ready) THEN
	IF NOT(GVL.s3363[s3363_Mapping.ACV_101].Ready) 		THEN	tStatus:=ez100_Status.ACV101_Not_Ready;END_IF;
	IF NOT(GVL.s3363[s3363_Mapping.ACV_102].Ready) 		THEN	tStatus:=ez100_Status.ACV102_Not_Ready;END_IF;
END_IF;

IF NOT(PVL.s8312[s8312_mapping.PT_101].Ready) 		THEN 	tStatus:=eZ100_Status.PT101_Not_Ready; END_IF;
IF NOT(PVL.s8098[s8098_Mapping.FT_101].Ready)		THEN	tStatus:=eZ100_Status.FT101_Not_Ready; END_IF;


IF GVL.LS[LS_Mapping.LSHH_201].Status.eStatus= Burkert.DI_Status.Liquid_Detected_Alarm THEN tStatus:=eZ100_Status.EP101_LSHH201_High_High_Level_Alarm; END_IF;
//IF PVL.AIT[AIT_Mapping.LT_01A].Status.eStatus=Burkert.eSensor_Status.Low_Low_Alarm THEN tStatus:=eZ100_Status.LT01A_Low_Low_Level_Alarm; END_IF;
//IF PVL.AIT[AIT_Mapping.LT_01B].Status.eStatus=Burkert.eSensor_Status.Low_Low_Alarm THEN tStatus:=eZ100_Status.LT01B_Low_Low_Level_Alarm; END_IF;
IF PVL.s8312[s8312_Mapping.PT_101].Status.eStatus=Burkert.eSensor_Status.Low_Low_Alarm THEN tStatus:=eZ100_Status.PT101_Low_Low_Pressure_Alarm; END_IF;
IF PVL.s8312[s8312_Mapping.PT_101].Status.eStatus=Burkert.eSensor_Status.HiHi_Alarm THEN tStatus:=eZ100_Status.PT101_High_High_Pressure_Alarm; END_IF;

IF PVl.Duplex[Duplex_mapping.Z100].Mode.eMode=Burkert.eDuplex_Mode.Disabled THEN	tStatus:=eZ100_Status.Pump_Duplex_Disabled; END_IF;


IF NOT(PVL.s8098[s8098_mapping.FT_101].Ready)	THEN	tStatus:=eZ100_Status.FT01_Not_Ready; END_IF;
IF PVl.s8098[s8098_mapping.FT_101].PDO.VolumeFlow.Status.eStatus=Burkert.eSensor_Status.Low_Low_Alarm THEN tStatus:=eZ100_Status.FT101_Low_Low_Flow_Alarm; END_IF;


PVl.Z100_Config.Status.eStatus:=tStatus;




              
END_ACTION

ACTION Evaluate_Level:
                tStatus:=Local_status;

//IF NOT(pvl.AIT[AIT_Mapping.LT_01A].Ready) 	THEN tStatus:=eZ100_Status.LT01A_Not_Ready; END_IF;
//IF NOT(pvl.AIT[AIT_Mapping.LT_01B].Ready) 	THEN tStatus:=eZ100_Status.LT01B_Not_Ready; END_IF;
IF NOT(pvl.AIT[AIT_Mapping.LT_101_P].Ready) 	THEN tStatus:=eZ100_Status.LT101_Not_Ready; END_IF;
IF PVL.AIT[AIT_Mapping.LT_101_P].Status.eStatus=Burkert.eSensor_Status.HiHi_Alarm THEN	tStatus:=eZ100_Status.EP101_LT101_High_High_Level_Alarm; END_IF;

IF NOT(PVL.AIT[AIT_Mapping.FT_01].Ready) 	THEN tStatus:=eZ100_Status.FT01_Not_Ready; END_IF;
IF GVL.LS[LS_Mapping.LSLL_101].Status.eStatus=Burkert.DI_Status.No_Liquid_Detected_Alarm THEN	tStatus:=eZ100_Status.LSLL101_Pump_Intakes_Dry; END_IF;
IF NOT(Network.VFD[VFD_Mapping.VFD_101A].Ready) AND NOT(Network.VFD[VFD_Mapping.VFD_101B].Ready) THEN
	IF NOT(Network.VFD[VFD_Mapping.VFD_101A].Ready)	 	THEN	tStatus:=eZ100_Status.Pump_101A_Not_Ready; END_IF;
	IF NOT(Network.VFD[VFD_Mapping.VFD_101B].Ready) 	THEN	tStatus:=eZ100_Status.Pump_101B_Not_Ready; END_IF;
END_IF;
IF NOT(GVL.s3363[s3363_Mapping.ACV_101].Ready) AND NOT(GVL.s3363[s3363_Mapping.ACV_102].Ready) THEN
	IF NOT(GVL.s3363[s3363_Mapping.ACV_101].Ready) 		THEN	tStatus:=ez100_Status.ACV101_Not_Ready;END_IF;
	IF NOT(GVL.s3363[s3363_Mapping.ACV_102].Ready) 		THEN	tStatus:=ez100_Status.ACV102_Not_Ready;END_IF;
END_IF;
IF NOT(PVL.s8312[s8312_mapping.PT_101].Ready) 		THEN 	tStatus:=eZ100_Status.PT101_Not_Ready; END_IF;
IF NOT(PVL.s8098[s8098_Mapping.FT_101].Ready)		THEN	tStatus:=eZ100_Status.FT101_Not_Ready; END_IF;


IF GVL.LS[LS_Mapping.LSHH_201].Status.eStatus= Burkert.DI_Status.Liquid_Detected_Alarm THEN tStatus:=eZ100_Status.EP101_LSHH201_High_High_Level_Alarm; END_IF;
//IF PVL.AIT[AIT_Mapping.LT_01A].Status.eStatus=Burkert.eSensor_Status.Low_Low_Alarm THEN tStatus:=eZ100_Status.LT01A_Low_Low_Level_Alarm; END_IF;
//IF PVL.AIT[AIT_Mapping.LT_01B].Status.eStatus=Burkert.eSensor_Status.Low_Low_Alarm THEN tStatus:=eZ100_Status.LT01B_Low_Low_Level_Alarm; END_IF;
IF PVL.s8312[s8312_Mapping.PT_101].Status.eStatus=Burkert.eSensor_Status.Low_Low_Alarm THEN tStatus:=eZ100_Status.PT101_Low_Low_Pressure_Alarm; END_IF;
IF PVL.s8312[s8312_Mapping.PT_101].Status.eStatus=Burkert.eSensor_Status.HiHi_Alarm THEN tStatus:=eZ100_Status.PT101_High_High_Pressure_Alarm; END_IF;


IF PVl.Duplex[Duplex_mapping.Z100].Mode.eMode=Burkert.eDuplex_Mode.Disabled THEN	tStatus:=eZ100_Status.Pump_Duplex_Disabled; END_IF;

IF NOT(PVL.s8098[s8098_mapping.FT_101].Ready)	THEN	tStatus:=eZ100_Status.FT01_Not_Ready; END_IF;
IF PVl.s8098[s8098_mapping.FT_101].PDO.VolumeFlow.Status.eStatus=Burkert.eSensor_Status.Low_Low_Alarm THEN tStatus:=eZ100_Status.FT101_Low_Low_Flow_Alarm; END_IF;

PVl.Z100_Config.Status.eStatus:=tStatus;




              
END_ACTION

ACTION Evaluate_Flow_Intake:
                tStatus:=Local_status;

//IF NOT(pvl.AIT[AIT_Mapping.LT_01A].Ready) 	THEN tStatus:=eZ100_Status.LT01A_Not_Ready; END_IF;
//IF NOT(pvl.AIT[AIT_Mapping.LT_01B].Ready) 	THEN tStatus:=eZ100_Status.LT01B_Not_Ready; END_IF;
IF NOT(pvl.AIT[AIT_Mapping.LT_101_P].Ready) 	THEN tStatus:=eZ100_Status.LT101_Not_Ready; END_IF;
IF PVL.AIT[AIT_Mapping.LT_101_P].Status.eStatus=Burkert.eSensor_Status.HiHi_Alarm THEN	tStatus:=eZ100_Status.EP101_LT101_High_High_Level_Alarm; END_IF;

//IF NOT(PVL.AIT[AIT_Mapping.FT_01].Ready) 	THEN tStatus:=eZ100_Status.FT01_Not_Ready; END_IF;
IF GVL.LS[LS_Mapping.LSLL_101].Status.eStatus=Burkert.DI_Status.No_Liquid_Detected_Alarm THEN	tStatus:=eZ100_Status.LSLL101_Pump_Intakes_Dry; END_IF;

IF NOT(Network.VFD[VFD_Mapping.VFD_101A].Ready) AND NOT(Network.VFD[VFD_Mapping.VFD_101B].Ready) THEN
	IF NOT(Network.VFD[VFD_Mapping.VFD_101A].Ready)	 	THEN	tStatus:=eZ100_Status.Pump_101A_Not_Ready; END_IF;
	IF NOT(Network.VFD[VFD_Mapping.VFD_101B].Ready) 	THEN	tStatus:=eZ100_Status.Pump_101B_Not_Ready; END_IF;
END_IF;
IF NOT(GVL.s3363[s3363_Mapping.ACV_101].Ready) AND NOT(GVL.s3363[s3363_Mapping.ACV_102].Ready) THEN
	IF NOT(GVL.s3363[s3363_Mapping.ACV_101].Ready) 		THEN	tStatus:=ez100_Status.ACV101_Not_Ready;END_IF;
	IF NOT(GVL.s3363[s3363_Mapping.ACV_102].Ready) 		THEN	tStatus:=ez100_Status.ACV102_Not_Ready;END_IF;
END_IF;
IF NOT(PVL.s8312[s8312_mapping.PT_101].Ready) 		THEN 	tStatus:=eZ100_Status.PT101_Not_Ready; END_IF;
IF NOT(PVL.s8098[s8098_Mapping.FT_101].Ready)		THEN	tStatus:=eZ100_Status.FT101_Not_Ready; END_IF;


IF GVL.LS[LS_Mapping.LSHH_201].Status.eStatus= Burkert.DI_Status.Liquid_Detected_Alarm THEN tStatus:=eZ100_Status.EP101_LSHH201_High_High_Level_Alarm; END_IF;
//IF PVL.AIT[AIT_Mapping.LT_01A].Status.eStatus=Burkert.eSensor_Status.Low_Low_Alarm THEN tStatus:=eZ100_Status.LT01A_Low_Low_Level_Alarm; END_IF;
//IF PVL.AIT[AIT_Mapping.LT_01B].Status.eStatus=Burkert.eSensor_Status.Low_Low_Alarm THEN tStatus:=eZ100_Status.LT01B_Low_Low_Level_Alarm; END_IF;
IF PVL.s8312[s8312_Mapping.PT_101].Status.eStatus=Burkert.eSensor_Status.Low_Low_Alarm THEN tStatus:=eZ100_Status.PT101_Low_Low_Pressure_Alarm; END_IF;
IF PVL.s8312[s8312_Mapping.PT_101].Status.eStatus=Burkert.eSensor_Status.HiHi_Alarm THEN tStatus:=eZ100_Status.PT101_High_High_Pressure_Alarm; END_IF;

IF NOT(PVL.s8098[s8098_mapping.FT_101].Ready)	THEN	tStatus:=eZ100_Status.FT01_Not_Ready; END_IF;
IF PVl.s8098[s8098_mapping.FT_101].PDO.VolumeFlow.Status.eStatus=Burkert.eSensor_Status.Low_Low_Alarm THEN tStatus:=eZ100_Status.FT101_Low_Low_Flow_Alarm; END_IF;


IF PVl.Duplex[Duplex_mapping.Z100].Mode.eMode=Burkert.eDuplex_Mode.Disabled THEN	tStatus:=eZ100_Status.Pump_Duplex_Disabled; END_IF;



PVl.Z100_Config.Status.eStatus:=tStatus;




              
END_ACTION

ACTION ACV_Manager:
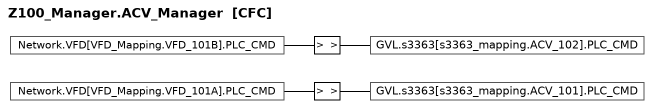
(* CFC diagram, written out as Structured Text *)
GVL.s3363[s3363_mapping.ACV_102].PLC_CMD := Network.VFD[VFD_Mapping.VFD_101B].PLC_CMD;
GVL.s3363[s3363_mapping.ACV_101].PLC_CMD := Network.VFD[VFD_Mapping.VFD_101A].PLC_CMD;
END_ACTION

ACTION Task_Flow_Discharge:
                IF PVL.Z100_Config.Task.eTask<> Local_Task THEN
	Local_Task:=PVL.Z100_Config.Task.eTask;
	local_status:=eZ100_Status.Flow_Control_Transfer;
	PVL.Z100_Config.READY:=TRUE;
END_IF;







PVL.PID[PID_Mapping.Z100_Flow].PLC_Target:=PVL.Z100_Config.Target_Flow.Target;
Burkert.Alarm_Window_Convert(window:=PVL.Z100_Config.Target_Flow,Config:=PVL.s8098[s8098_Mapping.FT_101].PDO.VolumeFlow.Alarm_Config);
Evaluate_Flow_Discharge();


CASE PVL.Z100_Config.Status.eStatus OF
	eZ100_Status.EP101_LSHH201_High_High_Level_Alarm: 		Local_Status:=PVL.Z100_Config.Status.eStatus; PVL.Z100_Config.READY:=FALSE;
	//eZ100_Status.EP101_LT101_High_High_Level_Alarm:			Local_Status:=PVL.Z100_Config.Status.eStatus;
	//eZ100_Status.LT01A_Low_Low_Level_Alarm:				Local_Status:=PVL.Z100_Config.Status.eStatus;
	//eZ100_Status.LT01B_Low_Low_Level_Alarm:				Local_Status:=PVL.Z100_Config.Status.eStatus;
	eZ100_Status.PT101_High_High_Pressure_Alarm:			Local_Status:=PVL.Z100_Config.Status.eStatus;PVL.Z100_Config.READY:=FALSE;
	eZ100_Status.PT101_Low_Low_Pressure_Alarm:				Local_Status:=PVL.Z100_Config.Status.eStatus;;PVL.Z100_Config.READY:=FALSE;
	eZ100_Status.LSLL101_Pump_Intakes_Dry:					Local_Status:=PVL.Z100_Config.Status.eStatus;PVL.Z100_Config.READY:=FALSE;
	eZ100_Status.FT101_Low_Low_Flow_Alarm:					Local_Status:=PVL.Z100_Config.Status.eStatus;PVL.Z100_Config.READY:=FALSE;
	
	eZ100_Status.LT101_High_High_Alarm:	PVL.Z100_Config.READY:=FALSE;
		IF PVl.AIT[ait_mapping.LT_101_P].Status.eStatus=Burkert.eSensor_Status.HiHi_Alarm THEN	
			Local_Status:=PVL.Z100_Config.Status.eStatus;
		ELSE
			Local_Status:=eZ100_Status.Waiting_For_Level_OK_LT101;
		END_IF
	eZ100_Status.Waiting_For_Level_OK_LT101: 
		PVL.Z100_Config.READY:=FALSE;
		IF PVl.AIT[ait_mapping.LT_101_P].Status.eStatus=Burkert.eSensor_Status.OK	THEN local_Task:=99; END_IF;
	
	eZ100_Status.Flow_Control_Transfer:	PVL.Z100_Config.READY:=TRUE;
	

END_CASE;
              
END_ACTION

ACTION Alarms:
                
CASE PVL.Z100_Config.Task.eTask OF

	eZ100_task.Off:	
		PVL.AIT[AIT_Mapping.LT_01A].Alarm_Config.Silence:=FALSE;
		PVL.AIT[AIT_Mapping.LT_01B].Alarm_Config.Silence:=FALSE;
		PVL.AIT[AIT_Mapping.FT_01].Alarm_Config.Silence:=TRUE;
		PVL.s8312[s8312_Mapping.PT_101].Alarm_Config.Silence:=TRUE;//TRUE;
		PVL.s8098[s8098_mapping.FT_101].PDO.VolumeFlow.Alarm_Config.Silence:=TRUE;
		PVL.s8098[s8098_mapping.FT_101].PDO.Temp.Alarm_Config.Silence:=TRUE;
		PVL.s8098[s8098_mapping.FT_101].PDO.Totaliser_1 .Alarm_Config.Silence:=TRUE;
		
	eZ100_Task.Batch:
		PVL.AIT[AIT_Mapping.LT_01A].Alarm_Config.Silence:=FALSE;
		PVL.AIT[AIT_Mapping.LT_01B].Alarm_Config.Silence:=FALSE;
		PVL.AIT[AIT_Mapping.FT_01].Alarm_Config.Silence:=FALSE;
		PVL.s8312[s8312_Mapping.PT_101].Alarm_Config.Silence:=(Network.VFD[VFD_Mapping.VFD_101A].Output_Pct<10 AND Network.VFD[VFD_Mapping.VFD_101B].Output_Pct<10);
		PVL.s8098[s8098_mapping.FT_101].PDO.VolumeFlow.Alarm_Config.Silence:=(Network.VFD[VFD_Mapping.VFD_101A].Output_Pct<10 AND Network.VFD[VFD_Mapping.VFD_101B].Output_Pct<10);
		PVL.s8098[s8098_mapping.FT_101].PDO.Temp.Alarm_Config.Silence:=FALSE;
		PVL.s8098[s8098_mapping.FT_101].PDO.Totaliser_1 .Alarm_Config.Silence:=(Network.VFD[VFD_Mapping.VFD_101A].Output_Pct<10 AND Network.VFD[VFD_Mapping.VFD_101B].Output_Pct<10);
	ez100_Task.Batch_Level:
		PVL.AIT[AIT_Mapping.LT_01A].Alarm_Config.Silence:=FALSE;
		PVL.AIT[AIT_Mapping.LT_01B].Alarm_Config.Silence:=FALSE;
		PVL.AIT[AIT_Mapping.FT_01].Alarm_Config.Silence:=FALSE;
		PVL.s8312[s8312_Mapping.PT_101].Alarm_Config.Silence:=(Network.VFD[VFD_Mapping.VFD_101A].Output_Pct<10 AND Network.VFD[VFD_Mapping.VFD_101B].Output_Pct<10);
		PVL.s8098[s8098_mapping.FT_101].PDO.VolumeFlow.Alarm_Config.Silence:=(Network.VFD[VFD_Mapping.VFD_101A].Output_Pct<10 AND Network.VFD[VFD_Mapping.VFD_101B].Output_Pct<10);
		PVL.s8098[s8098_mapping.FT_101].PDO.Temp.Alarm_Config.Silence:=FALSE;
		PVL.s8098[s8098_mapping.FT_101].PDO.Totaliser_1 .Alarm_Config.Silence:=(Network.VFD[VFD_Mapping.VFD_101A].Output_Pct<10 AND Network.VFD[VFD_Mapping.VFD_101B].Output_Pct<10);
	eZ100_Task.Continuous_Flow_Discharge:
		PVL.AIT[AIT_Mapping.LT_01A].Alarm_Config.Silence:=FALSE;
		PVL.AIT[AIT_Mapping.LT_01B].Alarm_Config.Silence:=FALSE;
		PVL.AIT[AIT_Mapping.FT_01].Alarm_Config.Silence:=FALSE;
		PVL.s8312[s8312_Mapping.PT_101].Alarm_Config.Silence:=(Network.VFD[VFD_Mapping.VFD_101A].Output_Pct<10 AND Network.VFD[VFD_Mapping.VFD_101B].Output_Pct<10);
		PVL.s8098[s8098_mapping.FT_101].PDO.VolumeFlow.Alarm_Config.Silence:=(Network.VFD[VFD_Mapping.VFD_101A].Output_Pct<10 AND Network.VFD[VFD_Mapping.VFD_101B].Output_Pct<10);
		PVL.s8098[s8098_mapping.FT_101].PDO.Temp.Alarm_Config.Silence:=FALSE;
		PVL.s8098[s8098_mapping.FT_101].PDO.Totaliser_1 .Alarm_Config.Silence:=(Network.VFD[VFD_Mapping.VFD_101A].Output_Pct<10 AND Network.VFD[VFD_Mapping.VFD_101B].Output_Pct<10);
	eZ100_Task.Continuous_Flow_Intake:
		PVL.AIT[AIT_Mapping.LT_01A].Alarm_Config.Silence:=FALSE;
		PVL.AIT[AIT_Mapping.LT_01B].Alarm_Config.Silence:=FALSE;
		PVL.AIT[AIT_Mapping.FT_01].Alarm_Config.Silence:=FALSE;
		PVL.s8312[s8312_Mapping.PT_101].Alarm_Config.Silence:=(Network.VFD[VFD_Mapping.VFD_101A].Output_Pct<10 AND Network.VFD[VFD_Mapping.VFD_101B].Output_Pct<10);
		PVL.s8098[s8098_mapping.FT_101].PDO.VolumeFlow.Alarm_Config.Silence:=(Network.VFD[VFD_Mapping.VFD_101A].Output_Pct<10 AND Network.VFD[VFD_Mapping.VFD_101B].Output_Pct<10);;
		PVL.s8098[s8098_mapping.FT_101].PDO.Temp.Alarm_Config.Silence:=FALSE;
		PVL.s8098[s8098_mapping.FT_101].PDO.Totaliser_1 .Alarm_Config.Silence:=(Network.VFD[VFD_Mapping.VFD_101A].Output_Pct<10 AND Network.VFD[VFD_Mapping.VFD_101B].Output_Pct<10);
	eZ100_Task.Continuous_Level:
		PVL.AIT[AIT_Mapping.LT_01A].Alarm_Config.Silence:=FALSE;
		PVL.AIT[AIT_Mapping.LT_01B].Alarm_Config.Silence:=FALSE;
		PVL.AIT[AIT_Mapping.FT_01].Alarm_Config.Silence:=FALSE;
		PVL.s8312[s8312_Mapping.PT_101].Alarm_Config.Silence:=(Network.VFD[VFD_Mapping.VFD_101A].Output_Pct<10 AND Network.VFD[VFD_Mapping.VFD_101B].Output_Pct<10);
		PVL.s8098[s8098_mapping.FT_101].PDO.VolumeFlow.Alarm_Config.Silence:=(Network.VFD[VFD_Mapping.VFD_101A].Output_Pct<10 AND Network.VFD[VFD_Mapping.VFD_101B].Output_Pct<10);
		PVL.s8098[s8098_mapping.FT_101].PDO.Temp.Alarm_Config.Silence:=FALSE;
		PVL.s8098[s8098_mapping.FT_101].PDO.Totaliser_1 .Alarm_Config.Silence:=(Network.VFD[VFD_Mapping.VFD_101A].Output_Pct<10 AND Network.VFD[VFD_Mapping.VFD_101B].Output_Pct<10);
	eZ100_Task.Continuous_UV:
		PVL.AIT[AIT_Mapping.LT_01A].Alarm_Config.Silence:=FALSE;
		PVL.AIT[AIT_Mapping.LT_01B].Alarm_Config.Silence:=FALSE;
		PVL.AIT[AIT_Mapping.FT_01].Alarm_Config.Silence:=FALSE;
		PVL.s8312[s8312_Mapping.PT_101].Alarm_Config.Silence:=(Network.VFD[VFD_Mapping.VFD_101A].Output_Pct<10 AND Network.VFD[VFD_Mapping.VFD_101B].Output_Pct<10);;
		PVL.s8098[s8098_mapping.FT_101].PDO.VolumeFlow.Alarm_Config.Silence:=FALSE;
		PVL.s8098[s8098_mapping.FT_101].PDO.Temp.Alarm_Config.Silence:=FALSE;
		PVL.s8098[s8098_mapping.FT_101].PDO.Totaliser_1 .Alarm_Config.Silence:=FALSE;
	eZ100_Task.Drain:
		PVL.AIT[AIT_Mapping.LT_01A].Alarm_Config.Silence:=FALSE;
		PVL.AIT[AIT_Mapping.LT_01B].Alarm_Config.Silence:=FALSE;
		PVL.AIT[AIT_Mapping.FT_01].Alarm_Config.Silence:=FALSE;
		PVL.s8312[s8312_Mapping.PT_101].Alarm_Config.Silence:=Network.VFD[VFD_Mapping.VFD_101A].Actual<10 AND Network.VFD[VFD_Mapping.VFD_101B].Actual<10;
		PVL.s8098[s8098_mapping.FT_101].PDO.VolumeFlow.Alarm_Config.Silence:=(Network.VFD[VFD_Mapping.VFD_101A].Output_Pct<10 AND Network.VFD[VFD_Mapping.VFD_101B].Output_Pct<10);
		PVL.s8098[s8098_mapping.FT_101].PDO.Temp.Alarm_Config.Silence:=FALSE;
		PVL.s8098[s8098_mapping.FT_101].PDO.Totaliser_1 .Alarm_Config.Silence:=(Network.VFD[VFD_Mapping.VFD_101A].Output_Pct<10 AND Network.VFD[VFD_Mapping.VFD_101B].Output_Pct<10);
END_CASE;


              
END_ACTION

ACTION Task_OFF:
                IF PVL.Z100_Config.Task.eTask<> Local_Task THEN
	Local_Task:=PVL.Z100_Config.Task.eTask;
END_IF;






local_status:=eZ100_Status.Off;
Evaluate_All();

PVL.Z100_Config.READY:=(Local_Status=PVl.Z100_Config.Status.eStatus);
              
END_ACTION

ACTION Evaluate_Batch:
                tStatus:=Local_status;

//IF NOT(pvl.AIT[AIT_Mapping.LT_01A].Ready) 	THEN tStatus:=eZ100_Status.LT01A_Not_Ready; END_IF;
//IF NOT(pvl.AIT[AIT_Mapping.LT_01B].Ready) 	THEN tStatus:=eZ100_Status.LT01B_Not_Ready; END_IF;
IF NOT(pvl.AIT[AIT_Mapping.LT_101_P].Ready) 	THEN tStatus:=eZ100_Status.LT101_Not_Ready; END_IF;
IF PVL.AIT[AIT_Mapping.LT_101_P].Status.eStatus=Burkert.eSensor_Status.HiHi_Alarm THEN	tStatus:=eZ100_Status.EP101_LT101_High_High_Level_Alarm; END_IF;
//IF NOT(PVL.AIT[AIT_Mapping.FT_01].Ready) 	THEN tStatus:=eZ100_Status.FT01_Not_Ready; END_IF;
IF GVL.LS[LS_Mapping.LSLL_101].Status.eStatus=Burkert.DI_Status.No_Liquid_Detected_Alarm THEN	tStatus:=eZ100_Status.LSLL101_Pump_Intakes_Dry; END_IF;


IF NOT(Network.VFD[VFD_Mapping.VFD_101A].Ready) AND NOT(Network.VFD[VFD_Mapping.VFD_101B].Ready) THEN
	IF NOT(Network.VFD[VFD_Mapping.VFD_101A].Ready)	 	THEN	tStatus:=eZ100_Status.Pump_101A_Not_Ready; END_IF;
	IF NOT(Network.VFD[VFD_Mapping.VFD_101B].Ready) 	THEN	tStatus:=eZ100_Status.Pump_101B_Not_Ready; END_IF;
END_IF;
IF NOT(GVL.s3363[s3363_Mapping.ACV_101].Ready) AND NOT(GVL.s3363[s3363_Mapping.ACV_102].Ready) THEN
	IF NOT(GVL.s3363[s3363_Mapping.ACV_101].Ready) 		THEN	tStatus:=ez100_Status.ACV101_Not_Ready;END_IF;
	IF NOT(GVL.s3363[s3363_Mapping.ACV_102].Ready) 		THEN	tStatus:=ez100_Status.ACV102_Not_Ready;END_IF;
END_IF;
IF NOT(PVL.s8312[s8312_mapping.PT_101].Ready) 		THEN 	tStatus:=eZ100_Status.PT101_Not_Ready; END_IF;
IF NOT(PVL.s8098[s8098_Mapping.FT_101].Ready)		THEN	tStatus:=eZ100_Status.FT101_Not_Ready; END_IF;


IF GVL.LS[LS_Mapping.LSHH_201].Status.eStatus= Burkert.DI_Status.Liquid_Detected_Alarm THEN tStatus:=eZ100_Status.EP101_LSHH201_High_High_Level_Alarm; END_IF;
//IF PVL.AIT[AIT_Mapping.LT_01A].Status.eStatus=Burkert.eSensor_Status.Low_Low_Alarm THEN tStatus:=eZ100_Status.LT01A_Low_Low_Level_Alarm; END_IF;
//IF PVL.AIT[AIT_Mapping.LT_01B].Status.eStatus=Burkert.eSensor_Status.Low_Low_Alarm THEN tStatus:=eZ100_Status.LT01B_Low_Low_Level_Alarm; END_IF;
IF PVL.s8312[s8312_Mapping.PT_101].Status.eStatus=Burkert.eSensor_Status.Low_Low_Alarm THEN tStatus:=eZ100_Status.PT101_Low_Low_Pressure_Alarm; END_IF;
IF PVL.s8312[s8312_Mapping.PT_101].Status.eStatus=Burkert.eSensor_Status.HiHi_Alarm THEN tStatus:=eZ100_Status.PT101_High_High_Pressure_Alarm; END_IF;

IF PVl.Duplex[Duplex_mapping.Z100].Mode.eMode=Burkert.eDuplex_Mode.Disabled THEN	tStatus:=eZ100_Status.Pump_Duplex_Disabled; END_IF;

IF NOT(PVL.s8098[s8098_mapping.FT_101].Ready)	THEN	tStatus:=eZ100_Status.FT01_Not_Ready; END_IF;
IF PVl.s8098[s8098_mapping.FT_101].PDO.VolumeFlow.Status.eStatus=Burkert.eSensor_Status.Low_Low_Alarm THEN tStatus:=eZ100_Status.FT101_Low_Low_Flow_Alarm; END_IF;

PVl.Z100_Config.Status.eStatus:=tStatus;




              
END_ACTION

ACTION Task_Level:
                IF PVL.Z100_Config.Task.eTask<> Local_Task THEN
	Local_Task:=PVL.Z100_Config.Task.eTask;
END_IF;






local_status:=eZ100_Status.Level_Control_Transfer;
PVL.PID[PID_Mapping.Z100_Level].PLC_Target:=PVL.Z100_Config.Target_Level.Target;
Burkert.Alarm_Window_Convert(
	window:=PVL.Z100_Config.Target_Level,
	Config:=PVL.s8098[s8098_Mapping.FT_101].PDO.VolumeFlow.Alarm_Config);
Evaluate_Level();



CASE PVL.Z100_Config.Status.eStatus OF
	eZ100_Status.EP101_LSHH201_High_High_Level_Alarm: 		Local_Status:=PVL.Z100_Config.Status.eStatus;
	//eZ100_Status.EP101_LT101_High_High_Level_Alarm:			Local_Status:=PVL.Z100_Config.Status.eStatus;
	//eZ100_Status.LT01A_Low_Low_Level_Alarm:				Local_Status:=PVL.Z100_Config.Status.eStatus;
	//eZ100_Status.LT01B_Low_Low_Level_Alarm:				Local_Status:=PVL.Z100_Config.Status.eStatus;
	eZ100_Status.PT101_High_High_Pressure_Alarm:			Local_Status:=PVL.Z100_Config.Status.eStatus;
	eZ100_Status.PT101_Low_Low_Pressure_Alarm:			Local_Status:=PVL.Z100_Config.Status.eStatus;
	eZ100_Status.LSLL101_Pump_Intakes_Dry:					Local_Status:=PVL.Z100_Config.Status.eStatus;
	eZ100_Status.FT101_Low_Low_Flow_Alarm:					Local_Status:=PVL.Z100_Config.Status.eStatus;
	
	
		eZ100_Status.LT101_High_High_Alarm:	
		IF PVl.AIT[ait_mapping.LT_101_P].Status.eStatus=Burkert.eSensor_Status.HiHi_Alarm THEN	
			Local_Status:=PVL.Z100_Config.Status.eStatus;
		ELSE
			Local_Status:=eZ100_Status.Waiting_For_Level_OK_LT101;
		END_IF
	eZ100_Status.Waiting_For_Level_OK_LT101: IF PVl.AIT[ait_mapping.LT_101_P].Status.eStatus=Burkert.eSensor_Status.OK	THEN local_Task:=99; END_IF;

END_CASE;
              
END_ACTION

ACTION Evaluate_Flow_Discharge:
                tStatus:=Local_status;

//IF NOT(pvl.AIT[AIT_Mapping.LT_01A].Ready) 	THEN tStatus:=eZ100_Status.LT01A_Not_Ready; END_IF;
//IF NOT(pvl.AIT[AIT_Mapping.LT_01B].Ready) 	THEN tStatus:=eZ100_Status.LT01B_Not_Ready; END_IF;
IF NOT(pvl.AIT[AIT_Mapping.LT_101_P].Ready) 	THEN tStatus:=eZ100_Status.LT101_Not_Ready; END_IF;
IF PVL.AIT[AIT_Mapping.LT_101_P].Status.eStatus=Burkert.eSensor_Status.HiHi_Alarm THEN	tStatus:=eZ100_Status.EP101_LT101_High_High_Level_Alarm; END_IF;

//IF NOT(PVL.AIT[AIT_Mapping.FT_01].Ready) 	THEN tStatus:=eZ100_Status.FT01_Not_Ready; END_IF;
IF GVL.LS[LS_Mapping.LSLL_101].Status.eStatus=Burkert.DI_Status.No_Liquid_Detected_Alarm THEN	tStatus:=eZ100_Status.LSLL101_Pump_Intakes_Dry; END_IF;

IF NOT(Network.VFD[VFD_Mapping.VFD_101A].Ready) AND NOT(Network.VFD[VFD_Mapping.VFD_101B].Ready) THEN
	IF NOT(Network.VFD[VFD_Mapping.VFD_101A].Ready)	 	THEN	tStatus:=eZ100_Status.Pump_101A_Not_Ready; END_IF;
	IF NOT(Network.VFD[VFD_Mapping.VFD_101B].Ready) 	THEN	tStatus:=eZ100_Status.Pump_101B_Not_Ready; END_IF;
END_IF;
IF NOT(GVL.s3363[s3363_Mapping.ACV_101].Ready) AND NOT(GVL.s3363[s3363_Mapping.ACV_102].Ready) THEN
	IF NOT(GVL.s3363[s3363_Mapping.ACV_101].Ready) 		THEN	tStatus:=ez100_Status.ACV101_Not_Ready;END_IF;
	IF NOT(GVL.s3363[s3363_Mapping.ACV_102].Ready) 		THEN	tStatus:=ez100_Status.ACV102_Not_Ready;END_IF;
END_IF;

IF NOT(PVL.s8312[s8312_mapping.PT_101].Ready) 		THEN 	tStatus:=eZ100_Status.PT101_Not_Ready; END_IF;
IF NOT(PVL.s8098[s8098_Mapping.FT_101].Ready)		THEN	tStatus:=eZ100_Status.FT101_Not_Ready; END_IF;


IF GVL.LS[LS_Mapping.LSHH_201].Status.eStatus= Burkert.DI_Status.Liquid_Detected_Alarm THEN tStatus:=eZ100_Status.EP101_LSHH201_High_High_Level_Alarm; END_IF;
//IF PVL.AIT[AIT_Mapping.LT_01A].Status.eStatus=Burkert.eSensor_Status.Low_Low_Alarm THEN tStatus:=eZ100_Status.LT01A_Low_Low_Level_Alarm; END_IF;
//IF PVL.AIT[AIT_Mapping.LT_01B].Status.eStatus=Burkert.eSensor_Status.Low_Low_Alarm THEN tStatus:=eZ100_Status.LT01B_Low_Low_Level_Alarm; END_IF;
IF PVL.s8312[s8312_Mapping.PT_101].Status.eStatus=Burkert.eSensor_Status.Low_Low_Alarm THEN tStatus:=eZ100_Status.PT101_Low_Low_Pressure_Alarm; END_IF;
IF PVL.s8312[s8312_Mapping.PT_101].Status.eStatus=Burkert.eSensor_Status.HiHi_Alarm THEN tStatus:=eZ100_Status.PT101_High_High_Pressure_Alarm; END_IF;


IF PVl.Duplex[Duplex_mapping.Z100].Mode.eMode=Burkert.eDuplex_Mode.Disabled THEN	tStatus:=eZ100_Status.Pump_Duplex_Disabled; END_IF;

IF NOT(PVL.s8098[s8098_mapping.FT_101].Ready)	THEN	tStatus:=eZ100_Status.FT01_Not_Ready; END_IF;
IF PVl.s8098[s8098_mapping.FT_101].PDO.VolumeFlow.Status.eStatus=Burkert.eSensor_Status.Low_Low_Alarm THEN tStatus:=eZ100_Status.FT101_Low_Low_Flow_Alarm; END_IF;

PVl.Z100_Config.Status.eStatus:=tStatus;




              
END_ACTION

ACTION Evaluate_Drain:
                tStatus:=Local_status;

//IF NOT(pvl.AIT[AIT_Mapping.LT_01A].Ready) 	THEN tStatus:=eZ100_Status.LT01A_Not_Ready; END_IF;
//IF NOT(pvl.AIT[AIT_Mapping.LT_01B].Ready) 	THEN tStatus:=eZ100_Status.LT01B_Not_Ready; END_IF;
IF NOT(pvl.AIT[AIT_Mapping.LT_101_P].Ready) 	THEN tStatus:=eZ100_Status.LT101_Not_Ready; END_IF;
IF PVL.AIT[AIT_Mapping.LT_101_P].Status.eStatus=Burkert.eSensor_Status.HiHi_Alarm THEN	tStatus:=eZ100_Status.EP101_LT101_High_High_Level_Alarm; END_IF;

//IF NOT(PVL.AIT[AIT_Mapping.FT_01].Ready) 	THEN tStatus:=eZ100_Status.FT01_Not_Ready; END_IF;
IF GVL.LS[LS_Mapping.LSLL_101].Status.eStatus=Burkert.DI_Status.No_Liquid_Detected_Alarm THEN	tStatus:=eZ100_Status.Drain_Complete; END_IF;
IF NOT(Network.VFD[VFD_Mapping.VFD_101A].Ready) AND NOT(Network.VFD[VFD_Mapping.VFD_101B].Ready) THEN
	IF NOT(Network.VFD[VFD_Mapping.VFD_101A].Ready)	 	THEN	tStatus:=eZ100_Status.Pump_101A_Not_Ready; END_IF;
	IF NOT(Network.VFD[VFD_Mapping.VFD_101B].Ready) 	THEN	tStatus:=eZ100_Status.Pump_101B_Not_Ready; END_IF;
END_IF;
IF NOT(GVL.s3363[s3363_Mapping.ACV_101].Ready) AND NOT(GVL.s3363[s3363_Mapping.ACV_102].Ready) THEN
	IF NOT(GVL.s3363[s3363_Mapping.ACV_101].Ready) 		THEN	tStatus:=ez100_Status.ACV101_Not_Ready;END_IF;
	IF NOT(GVL.s3363[s3363_Mapping.ACV_102].Ready) 		THEN	tStatus:=ez100_Status.ACV102_Not_Ready;END_IF;
END_IF;
//IF NOT(PVL.s8312[s8312_mapping.PT_101].Ready) 		THEN 	tStatus:=eZ100_Status.PT101_Not_Ready; END_IF;
IF NOT(PVL.s8098[s8098_Mapping.FT_101].Ready)		THEN	tStatus:=eZ100_Status.FT101_Not_Ready; END_IF;


IF GVL.LS[LS_Mapping.LSHH_201].Status.eStatus= Burkert.DI_Status.Liquid_Detected_Alarm THEN tStatus:=eZ100_Status.EP101_LSHH201_High_High_Level_Alarm; END_IF;
//IF PVL.AIT[AIT_Mapping.LT_01A].Status.eStatus=Burkert.eSensor_Status.Low_Low_Alarm THEN tStatus:=eZ100_Status.LT01A_Low_Low_Level_Alarm; END_IF;
//IF PVL.AIT[AIT_Mapping.LT_01B].Status.eStatus=Burkert.eSensor_Status.Low_Low_Alarm THEN tStatus:=eZ100_Status.LT01B_Low_Low_Level_Alarm; END_IF;
IF PVL.s8312[s8312_Mapping.PT_101].Status.eStatus=Burkert.eSensor_Status.Low_Low_Alarm THEN tStatus:=eZ100_Status.PT101_Low_Low_Pressure_Alarm; END_IF;
IF PVL.s8312[s8312_Mapping.PT_101].Status.eStatus=Burkert.eSensor_Status.HiHi_Alarm THEN tStatus:=eZ100_Status.PT101_High_High_Pressure_Alarm; END_IF;


IF PVl.Duplex[Duplex_mapping.Z100].Mode.eMode=Burkert.eDuplex_Mode.Disabled THEN	tStatus:=eZ100_Status.Pump_Duplex_Disabled; END_IF;

IF NOT(PVL.s8098[s8098_mapping.FT_101].Ready)	THEN	tStatus:=eZ100_Status.FT01_Not_Ready; END_IF;
IF PVl.s8098[s8098_mapping.FT_101].PDO.VolumeFlow.Status.eStatus=Burkert.eSensor_Status.Low_Low_Alarm THEN tStatus:=eZ100_Status.FT101_Low_Low_Flow_Alarm; END_IF;

PVl.Z100_Config.Status.eStatus:=tStatus;




              
END_ACTION
END_PROGRAM

PROGRAM s336x_Manager
  VAR
    ACV_101_CTRL : Burkert.MbTCP_336x;
    ACV_102_CTRL : Burkert.MbTCP_336x;
    ACV_201_CTRL : Burkert.MbTCP_336x;
    ACV_203_CTRL : Burkert.MbTCP_336x;
    ACV_206_CTRL : Burkert.MbTCP_336x;
    ACV_207_CTRL : Burkert.MbTCP_336x;
    ACV_208_CTRL : Burkert.MbTCP_336x;
    ACV_209_CTRL : Burkert.MbTCP_336x;
    ACV_210_CTRL : Burkert.MbTCP_336x;
    ACV_213_CTRL : Burkert.MbTCP_336x;
    ACV_214_CTRL : Burkert.MbTCP_336x;
    ACV_215_CTRL : Burkert.MbTCP_336x;
    ACV_216_CTRL : Burkert.MbTCP_336x;
    ACV_219_CTRL : Burkert.MbTCP_336x;
    ACV_224_CTRL : Burkert.MbTCP_336x;
    ACV_225_CTRL : Burkert.MbTCP_336x;
    ACV_226_CTRL : Burkert.MbTCP_336x;
    Filter_Active : BOOL;
    Prerssure_Release : TOF;
  END_VAR
  VAR  (* added by the conversion: wires and edge detectors of the diagram *)
    _OR3_OUT : BOOL;
    _OR22_OUT : BOOL;
    _OR28_OUT : BOOL;
    _OR31_OUT : BOOL;
    _AND35_OUT : BOOL;
    _OR43_OUT : BOOL;
    _OR45_OUT : BOOL;
    _OR65_OUT : BOOL;
    _OR7_OUT : BOOL;
    _or9_OUT : BOOL;
    _OR5_OUT : BOOL;
    _OR3_OUT_2 : BOOL;
    _OR9_OUT_2 : BOOL;
    _OR7_OUT_2 : BOOL;
    _OR5_OUT_2 : BOOL;
    _OR11_OUT : BOOL;
  END_VAR

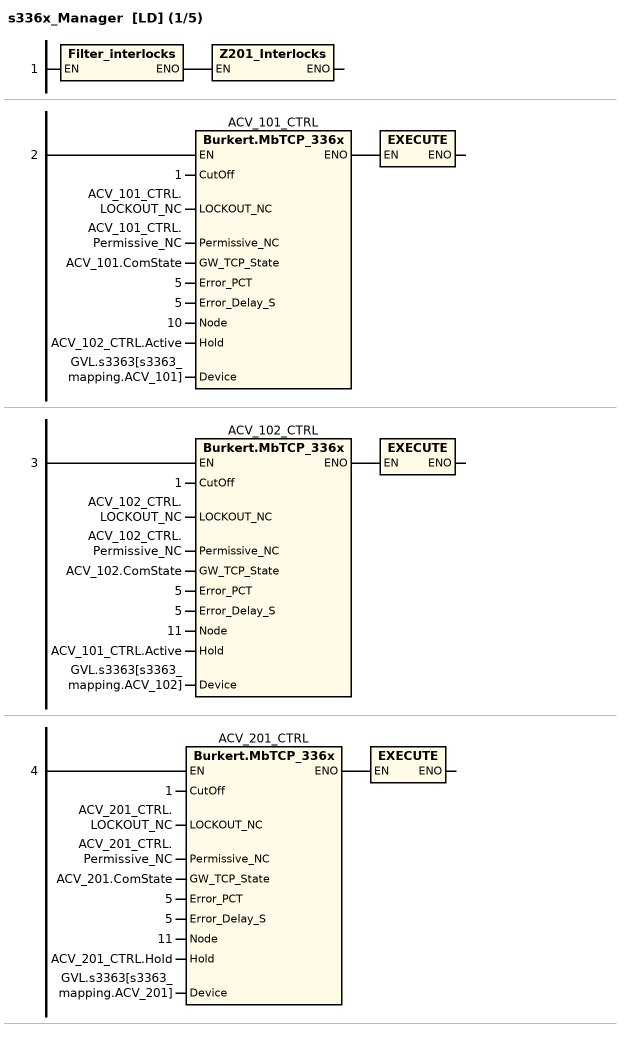
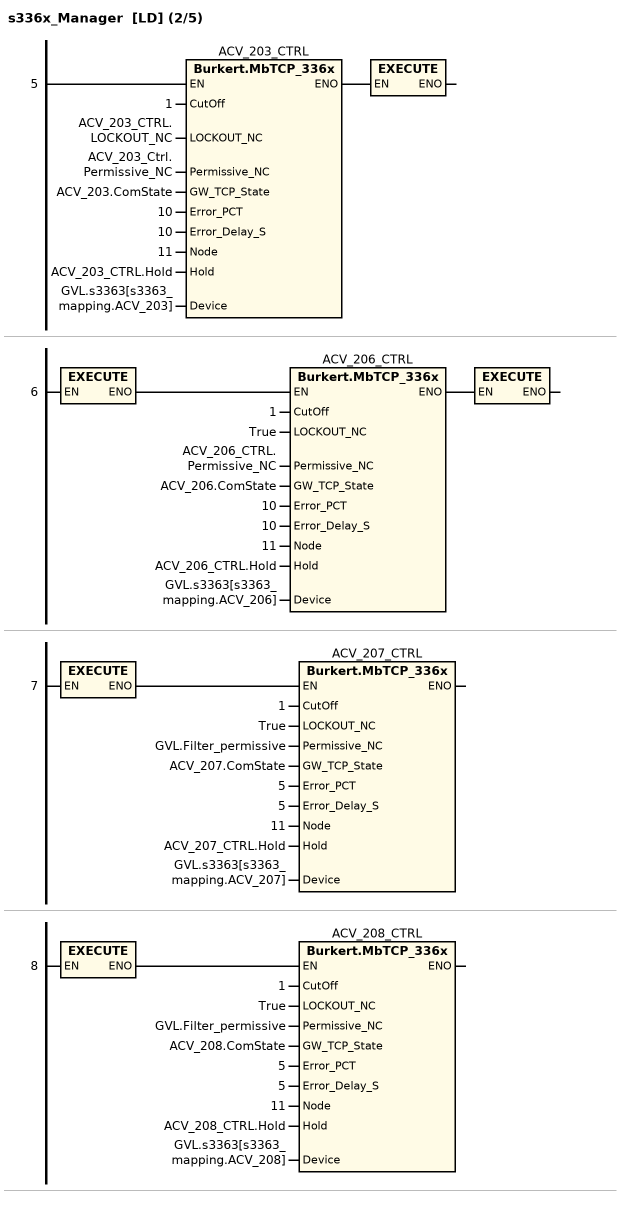
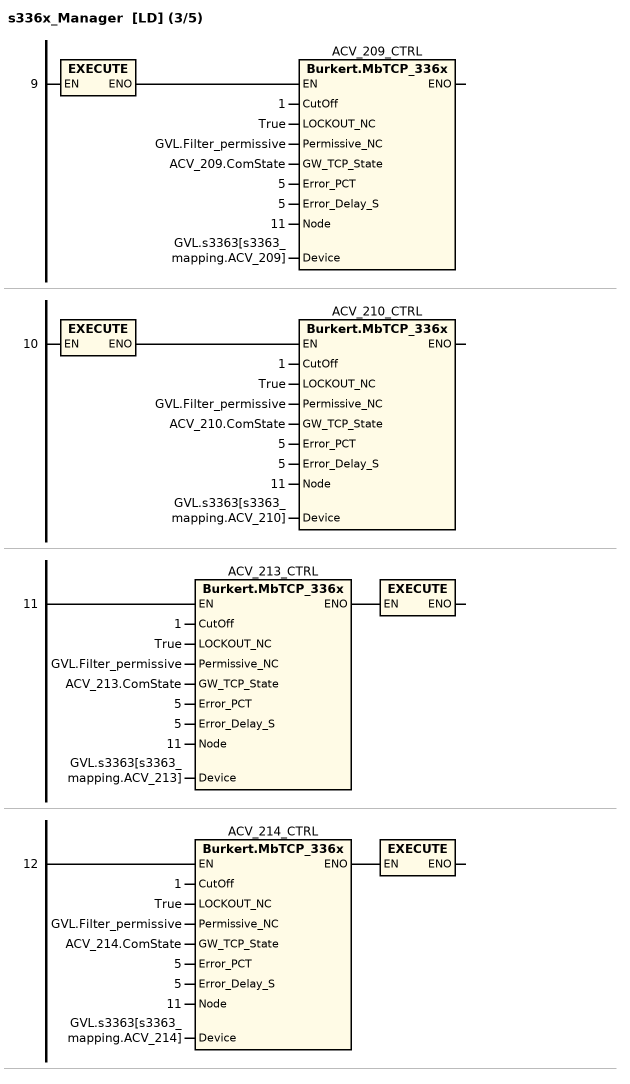
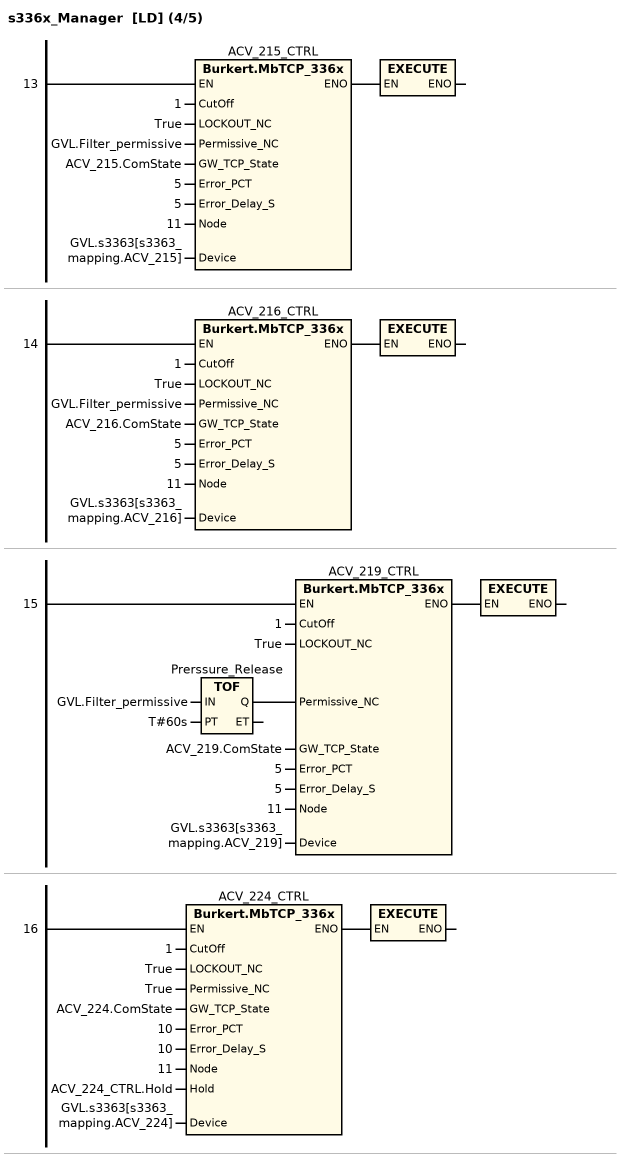
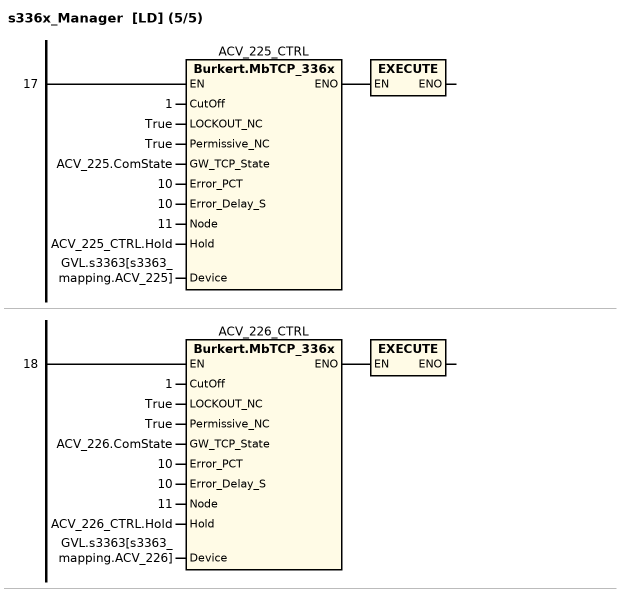
(* LD diagram, written out as Structured Text *)

Filter_interlocks();
Z201_Interlocks();

ACV_101_CTRL(CutOff := 1, LOCKOUT_NC := ACV_101_CTRL.LOCKOUT_NC, Permissive_NC := ACV_101_CTRL.Permissive_NC, GW_TCP_State := ACV_101.ComState, Error_PCT := 5, Error_Delay_S := 5, Node := 10, Hold := ACV_102_CTRL.Active, Device := GVL.s3363[s3363_mapping.ACV_101]);
IF ACV_101_CTRL.ENO THEN
  ACV_101_CTRL.Permissive_NC:=TRUE;
  ACV_101_CTRL.LOCKOUT_NC:= NOT(
  	GVL.LS[LS_Mapping.LSHH_201].Status.eStatus=Burkert.DI_Status.Liquid_Detected OR
  	GVL.LS[LS_Mapping.LSHH_201].Status.eStatus=Burkert.DI_Status.Liquid_Detected_Alarm
  	);
END_IF;

ACV_102_CTRL(CutOff := 1, LOCKOUT_NC := ACV_102_CTRL.LOCKOUT_NC, Permissive_NC := ACV_102_CTRL.Permissive_NC, GW_TCP_State := ACV_102.ComState, Error_PCT := 5, Error_Delay_S := 5, Node := 11, Hold := ACV_101_CTRL.Active, Device := GVL.s3363[s3363_mapping.ACV_102]);
IF ACV_102_CTRL.ENO THEN
  ACV_102_CTRL.Permissive_NC:=TRUE;
  ACV_102_CTRL.LOCKOUT_NC:= NOT(
  	GVL.LS[LS_Mapping.LSHH_201].Status.eStatus=Burkert.DI_Status.Liquid_Detected OR
  	GVL.LS[LS_Mapping.LSHH_201].Status.eStatus=Burkert.DI_Status.Liquid_Detected_Alarm
  	);
END_IF;


ACV_201_CTRL(CutOff := 1, LOCKOUT_NC := ACV_201_CTRL.LOCKOUT_NC, Permissive_NC := ACV_201_CTRL.Permissive_NC, GW_TCP_State := ACV_201.ComState, Error_PCT := 5, Error_Delay_S := 5, Node := 11, Hold := ACV_201_CTRL.Hold, Device := GVL.s3363[s3363_mapping.ACV_201]);
IF ACV_201_CTRL.ENO THEN
  ACV_201_CTRL.Permissive_NC:=TRUE;
  ACV_201_CTRL.LOCKOUT_NC:= (
  	NOT(GVL.LS[LS_Mapping.LSHH_204].Status.eStatus=Burkert.DI_Status.Liquid_Detected OR
  		GVL.LS[LS_Mapping.LSHH_204].Status.eStatus=Burkert.DI_Status.Liquid_Detected_Alarm)
  );
END_IF;


ACV_203_CTRL(CutOff := 1, LOCKOUT_NC := ACV_203_CTRL.LOCKOUT_NC, Permissive_NC := ACV_203_Ctrl.Permissive_NC, GW_TCP_State := ACV_203.ComState, Error_PCT := 10, Error_Delay_S := 10, Node := 11, Hold := ACV_203_CTRL.Hold, Device := GVL.s3363[s3363_mapping.ACV_203]);
IF ACV_203_CTRL.ENO THEN
  ACV_203_Ctrl.Permissive_NC:=TRUE;
  ACV_203_CTRL.LOCKOUT_NC:= NOT(
  	GVL.LS[LS_mapping.LSHH_201].Status.eStatus=Burkert.DI_Status.Liquid_Detected_Alarm OR
  	GVL.LS[LS_mapping.LSHH_201].Status.eStatus=Burkert.DI_Status.Liquid_Detected
  	);
END_IF;

(*ACV_206_CTRL.Hold:=(
	//ACV_206_CTRL.Active OR
	ACV_207_CTRL.Active OR
	ACV_208_CTRL.Active OR
	ACV_209_CTRL.Active OR
	ACV_210_CTRL.Active OR
	ACV_213_CTRL.Active OR
	ACV_214_CTRL.Active OR
	ACV_215_CTRL.Active OR
	ACV_216_CTRL.Active OR
	ACV_219_CTRL.Active
);*)
ACV_206_CTRL(CutOff := 1, LOCKOUT_NC := True, Permissive_NC := ACV_206_CTRL.Permissive_NC, GW_TCP_State := ACV_206.ComState, Error_PCT := 10, Error_Delay_S := 10, Node := 11, Hold := ACV_206_CTRL.Hold, Device := GVL.s3363[s3363_mapping.ACV_206]);
IF ACV_206_CTRL.ENO THEN
  IF (
  	PVl.Z202_Config.Task.eTask=eZ202_Task.Filter_Flow_P202_Recovery_Flow_P203 OR
  	PVl.Z202_Config.Task.eTask=eZ202_Task.Filter_Flow_P202_Recovery_Speed_P203 OR
  	PVl.Z202_Config.Task.eTask=eZ202_Task.Filter_Flow_P203 OR
  	PVl.Z202_Config.Task.eTask=eZ202_Task.Filter_Level_P202 OR
  	PVl.Z202_Config.Task.eTask=eZ202_Task.Filter_Level_P202_Recovery_Flow_P203 OR
  	PVl.Z202_Config.Task.eTask=eZ202_Task.Filter_Level_P202_Recovery_Speed_P203 OR
  	PVl.Z202_Config.Task.eTask=eZ202_Task.Filter_Level_P203) THEN
  
  
  	ACV_206_CTRL.Permissive_NC:=	GVL.Filter_permissive;
  ELSE
  	ACV_206_CTRL.Permissive_NC:=TRUE;
  END_IF
END_IF;

(*ACV_207_CTRL.Hold:=(
	ACV_206_CTRL.Active OR ACV_206_CTRL.Hold OR
	//ACV_207_CTRL.Active OR
	ACV_208_CTRL.Active OR
	ACV_209_CTRL.Active OR
	ACV_210_CTRL.Active OR
	ACV_213_CTRL.Active OR
	ACV_214_CTRL.Active OR
	ACV_215_CTRL.Active OR
	ACV_216_CTRL.Active OR
	ACV_219_CTRL.Active
);*)
ACV_207_CTRL(CutOff := 1, LOCKOUT_NC := True, Permissive_NC := GVL.Filter_permissive, GW_TCP_State := ACV_207.ComState, Error_PCT := 5, Error_Delay_S := 5, Node := 11, Hold := ACV_207_CTRL.Hold, Device := GVL.s3363[s3363_mapping.ACV_207]);

(*ACV_208_CTRL.Hold:=(
	ACV_206_CTRL.Active OR
	ACV_207_CTRL.Active OR ACV_207_CTRL.Hold OR
	//ACV_208_CTRL.Active OR
	ACV_209_CTRL.Active OR
	ACV_210_CTRL.Active OR
	ACV_213_CTRL.Active OR
	ACV_214_CTRL.Active OR
	ACV_215_CTRL.Active OR
	ACV_216_CTRL.Active OR
	ACV_219_CTRL.Active
);*)
ACV_208_CTRL(CutOff := 1, LOCKOUT_NC := True, Permissive_NC := GVL.Filter_permissive, GW_TCP_State := ACV_208.ComState, Error_PCT := 5, Error_Delay_S := 5, Node := 11, Hold := ACV_208_CTRL.Hold, Device := GVL.s3363[s3363_mapping.ACV_208]);

(*ACV_209_CTRL.Hold:=(
	ACV_206_CTRL.Active OR
	ACV_207_CTRL.Active OR
	ACV_208_CTRL.Active OR ACV_208_CTRL.Hold OR
	//ACV_209_CTRL.Active OR
	ACV_210_CTRL.Active OR
	ACV_213_CTRL.Active OR
	ACV_214_CTRL.Active OR
	ACV_215_CTRL.Active OR
	ACV_216_CTRL.Active OR
	ACV_219_CTRL.Active
);*)
ACV_209_CTRL(CutOff := 1, LOCKOUT_NC := True, Permissive_NC := GVL.Filter_permissive, GW_TCP_State := ACV_209.ComState, Error_PCT := 5, Error_Delay_S := 5, Node := 11, Device := GVL.s3363[s3363_mapping.ACV_209]);

(*ACV_210_CTRL.Hold:=(
	ACV_206_CTRL.Active OR
	ACV_207_CTRL.Active OR
	ACV_208_CTRL.Active OR
	ACV_209_CTRL.Active OR ACV_209_CTRL.Hold OR
	//ACV_210_CTRL.Active OR
	ACV_213_CTRL.Active OR
	ACV_214_CTRL.Active OR
	ACV_215_CTRL.Active OR
	ACV_216_CTRL.Active OR
	ACV_219_CTRL.Active
);*)
ACV_210_CTRL(CutOff := 1, LOCKOUT_NC := True, Permissive_NC := GVL.Filter_permissive, GW_TCP_State := ACV_210.ComState, Error_PCT := 5, Error_Delay_S := 5, Node := 11, Device := GVL.s3363[s3363_mapping.ACV_210]);

ACV_213_CTRL(CutOff := 1, LOCKOUT_NC := True, Permissive_NC := GVL.Filter_permissive, GW_TCP_State := ACV_213.ComState, Error_PCT := 5, Error_Delay_S := 5, Node := 11, Device := GVL.s3363[s3363_mapping.ACV_213]);
IF ACV_213_CTRL.ENO THEN EXECUTE(); END_IF;

ACV_214_CTRL(CutOff := 1, LOCKOUT_NC := True, Permissive_NC := GVL.Filter_permissive, GW_TCP_State := ACV_214.ComState, Error_PCT := 5, Error_Delay_S := 5, Node := 11, Device := GVL.s3363[s3363_mapping.ACV_214]);
IF ACV_214_CTRL.ENO THEN EXECUTE(); END_IF;

ACV_215_CTRL(CutOff := 1, LOCKOUT_NC := True, Permissive_NC := GVL.Filter_permissive, GW_TCP_State := ACV_215.ComState, Error_PCT := 5, Error_Delay_S := 5, Node := 11, Device := GVL.s3363[s3363_mapping.ACV_215]);
IF ACV_215_CTRL.ENO THEN EXECUTE(); END_IF;

ACV_216_CTRL(CutOff := 1, LOCKOUT_NC := True, Permissive_NC := GVL.Filter_permissive, GW_TCP_State := ACV_216.ComState, Error_PCT := 5, Error_Delay_S := 5, Node := 11, Device := GVL.s3363[s3363_mapping.ACV_216]);
IF ACV_216_CTRL.ENO THEN EXECUTE(); END_IF;

Prerssure_Release(IN := GVL.Filter_permissive, PT := T#60s);
ACV_219_CTRL(CutOff := 1, LOCKOUT_NC := True, Permissive_NC := Prerssure_Release.Q, GW_TCP_State := ACV_219.ComState, Error_PCT := 5, Error_Delay_S := 5, Node := 11, Device := GVL.s3363[s3363_mapping.ACV_219]);
IF ACV_219_CTRL.ENO THEN EXECUTE(); END_IF;

ACV_224_CTRL(CutOff := 1, LOCKOUT_NC := True, Permissive_NC := True, GW_TCP_State := ACV_224.ComState, Error_PCT := 10, Error_Delay_S := 10, Node := 11, Hold := ACV_224_CTRL.Hold, Device := GVL.s3363[s3363_mapping.ACV_224]);
IF ACV_224_CTRL.ENO THEN
  ACV_224_CTRL.Hold:=(
  	ACV_201_CTRL.Active OR
  	ACV_203_CTRL.Active OR
  	//ACV_224_CTRL.Active OR
  	ACV_225_CTRL.Active OR
  	ACV_226_CTRL.Active
  );
END_IF;

ACV_225_CTRL(CutOff := 1, LOCKOUT_NC := True, Permissive_NC := True, GW_TCP_State := ACV_225.ComState, Error_PCT := 10, Error_Delay_S := 10, Node := 11, Hold := ACV_225_CTRL.Hold, Device := GVL.s3363[s3363_mapping.ACV_225]);
IF ACV_225_CTRL.ENO THEN
  ACV_225_CTRL.Hold:=(
  	ACV_201_CTRL.Active OR
  	ACV_203_CTRL.Active OR
  	ACV_224_CTRL.Active OR
  	///ACV_225_CTRL.Active OR
  	ACV_226_CTRL.Active
  );
END_IF;

ACV_226_CTRL(CutOff := 1, LOCKOUT_NC := True, Permissive_NC := True, GW_TCP_State := ACV_226.ComState, Error_PCT := 10, Error_Delay_S := 10, Node := 11, Hold := ACV_226_CTRL.Hold, Device := GVL.s3363[s3363_mapping.ACV_226]);
IF ACV_226_CTRL.ENO THEN
  ACV_226_CTRL.Hold:=(
  	ACV_201_CTRL.Active OR
  	ACV_203_CTRL.Active OR
  	ACV_224_CTRL.Active OR
  	ACV_225_CTRL.Active //OR
  	//ACV_226_CTRL.Active
  );
END_IF;
(* --- network --- *)

ACTION Filter_Interlocks:
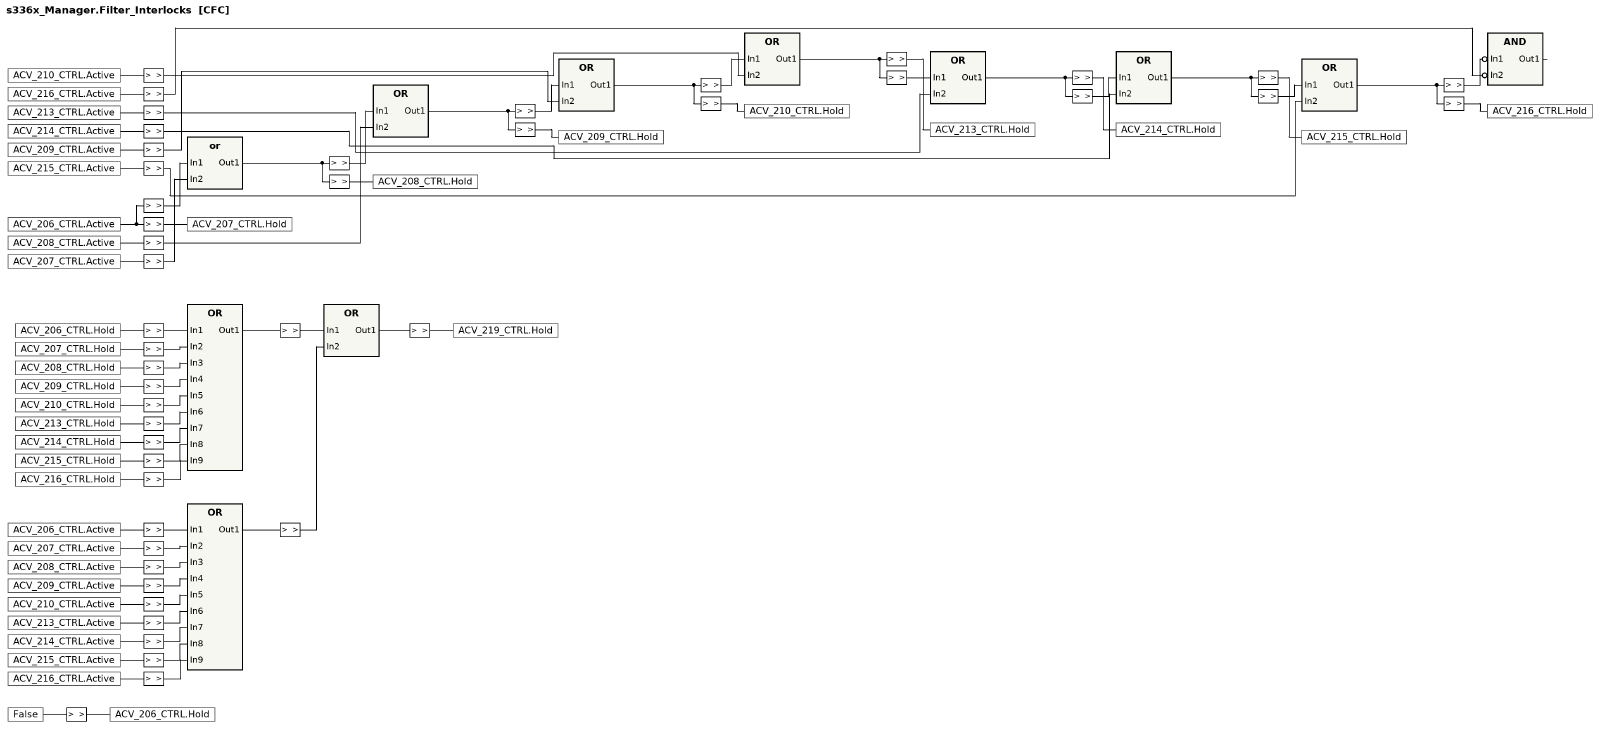
(* CFC diagram, written out as Structured Text *)
ACV_213_CTRL.Hold := _OR3_OUT;
ACV_214_CTRL.Hold := _OR22_OUT;
ACV_215_CTRL.Hold := _OR28_OUT;
_OR31_OUT := _OR28_OUT OR ACV_215_CTRL.Active;
_AND35_OUT := NOT _OR31_OUT AND NOT ACV_216_CTRL.Active;
ACV_216_CTRL.Hold := _OR31_OUT;
ACV_219_CTRL.Hold := _OR43_OUT;
_OR43_OUT := _OR45_OUT OR _OR65_OUT;
_OR65_OUT := ACV_206_CTRL.Active OR ACV_207_CTRL.Active OR ACV_208_CTRL.Active OR ACV_209_CTRL.Active OR ACV_210_CTRL.Active OR ACV_213_CTRL.Active OR ACV_214_CTRL.Active OR ACV_215_CTRL.Active OR ACV_216_CTRL.Active;
ACV_206_CTRL.Hold := False;
ACV_209_CTRL.Hold := _OR7_OUT;
ACV_208_CTRL.Hold := _or9_OUT;
ACV_210_CTRL.Hold := _OR5_OUT;
ACV_207_CTRL.Hold := ACV_206_CTRL.Active;
_or9_OUT := ACV_206_CTRL.Active OR ACV_207_CTRL.Active;
_OR7_OUT := _or9_OUT OR ACV_208_CTRL.Active;
_OR5_OUT := _OR7_OUT OR ACV_209_CTRL.Active;
_OR3_OUT := _OR5_OUT OR ACV_210_CTRL.Active;
_OR22_OUT := _OR3_OUT OR ACV_213_CTRL.Active;
_OR28_OUT := _OR22_OUT OR ACV_214_CTRL.Active;
_OR45_OUT := ACV_206_CTRL.Hold OR ACV_207_CTRL.Hold OR ACV_208_CTRL.Hold OR ACV_209_CTRL.Hold OR ACV_210_CTRL.Hold OR ACV_213_CTRL.Hold OR ACV_214_CTRL.Hold OR ACV_215_CTRL.Hold OR ACV_216_CTRL.Hold;
END_ACTION

ACTION Z201_Interlocks:
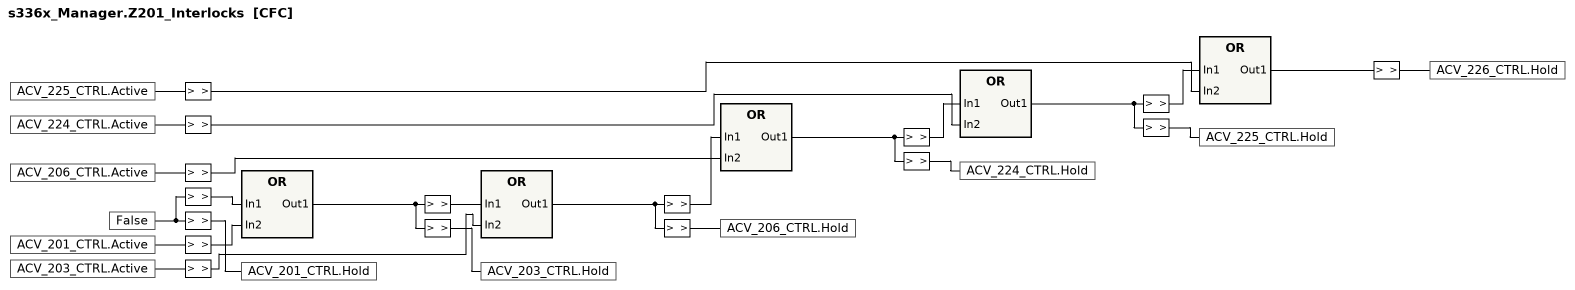
(* CFC diagram, written out as Structured Text *)
ACV_226_CTRL.Hold := _OR3_OUT_2;
ACV_206_CTRL.Hold := _OR9_OUT_2;
_OR7_OUT_2 := _OR9_OUT_2 OR ACV_206_CTRL.Active;
ACV_225_CTRL.Hold := _OR5_OUT_2;
_OR3_OUT_2 := _OR5_OUT_2 OR ACV_225_CTRL.Active;
ACV_201_CTRL.Hold := False;
ACV_203_CTRL.Hold := _OR11_OUT;
ACV_224_CTRL.Hold := _OR7_OUT_2;
_OR11_OUT := False OR ACV_201_CTRL.Active;
_OR9_OUT_2 := _OR11_OUT OR ACV_203_CTRL.Active;
_OR5_OUT_2 := _OR7_OUT_2 OR ACV_224_CTRL.Active;
END_ACTION
END_PROGRAM

PROGRAM ME44_IO
  VAR
    GW201_S2_Ready : BOOL;
  END_VAR

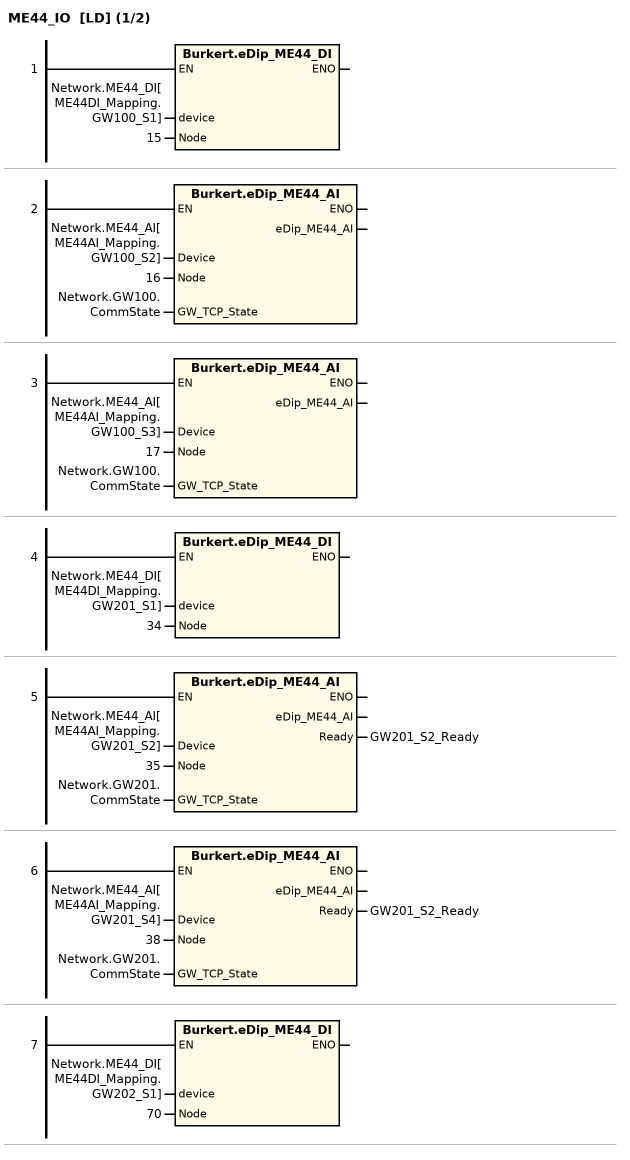
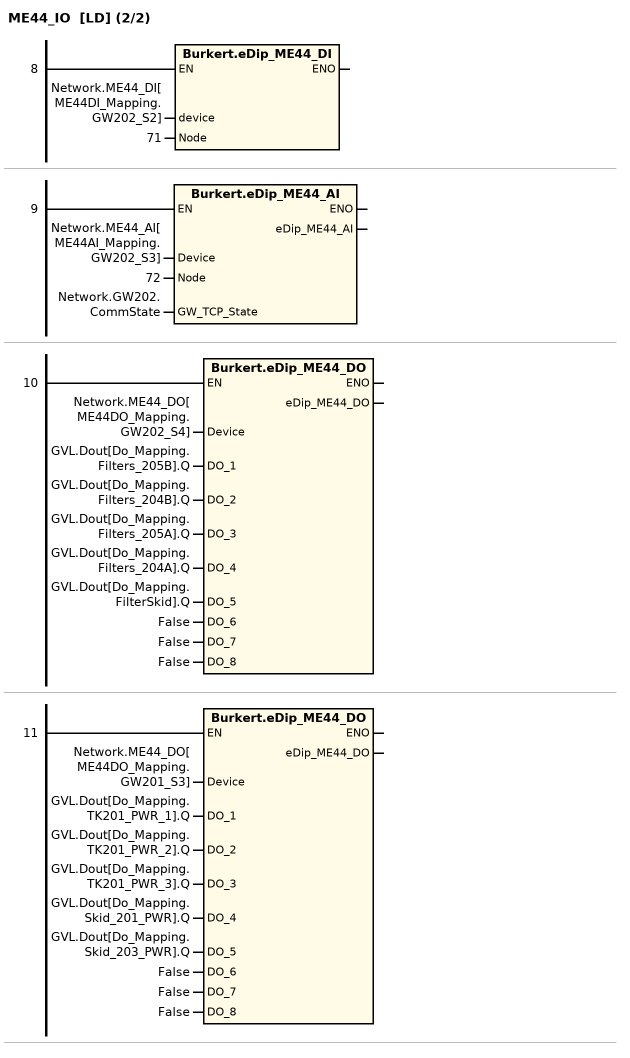
(* LD diagram, written out as Structured Text *)

Burkert.eDip_ME44_DI(Network.ME44_DI[ME44DI_Mapping.GW100_S1], 15);

Burkert.eDip_ME44_AI(Network.ME44_AI[ME44AI_Mapping. GW100_S2], 16, Network.GW100.CommState);

Burkert.eDip_ME44_AI(Network.ME44_AI[ME44AI_Mapping. GW100_S3], 17, Network.GW100.CommState);


Burkert.eDip_ME44_DI(Network.ME44_DI[ME44DI_Mapping.GW201_S1], 34);

Burkert.eDip_ME44_AI(Device := Network.ME44_AI[ME44AI_Mapping. GW201_S2], Node := 35, GW_TCP_State := Network.GW201.CommState, Ready => GW201_S2_Ready);

Burkert.eDip_ME44_AI(Device := Network.ME44_AI[ME44AI_Mapping. GW201_S4], Node := 38, GW_TCP_State := Network.GW201.CommState, Ready => GW201_S2_Ready);


Burkert.eDip_ME44_DI(Network.ME44_DI[ME44DI_Mapping.GW202_S1], 70);

Burkert.eDip_ME44_DI(Network.ME44_DI[ME44DI_Mapping.GW202_S2], 71);

Burkert.eDip_ME44_AI(Network.ME44_AI[ME44AI_Mapping. GW202_S3], 72, Network.GW202.CommState);

Burkert.eDip_ME44_DO(Network.ME44_DO[ME44DO_Mapping.GW202_S4], GVL.Dout[Do_Mapping.Filters_205B].Q, GVL.Dout[Do_Mapping.Filters_204B].Q, GVL.Dout[Do_Mapping.Filters_205A].Q, GVL.Dout[Do_Mapping.Filters_204A].Q, GVL.Dout[Do_Mapping.FilterSkid].Q, False, False, False);

Burkert.eDip_ME44_DO(Network.ME44_DO[ME44DO_Mapping.GW201_S3], GVL.Dout[Do_Mapping.TK201_PWR_1].Q, GVL.Dout[Do_Mapping.TK201_PWR_2].Q, GVL.Dout[Do_Mapping.TK201_PWR_3].Q, GVL.Dout[Do_Mapping.Skid_201_PWR].Q, GVL.Dout[Do_Mapping.Skid_203_PWR].Q, False, False, False);
(* --- network --- *)
END_PROGRAM

PROGRAM DO_Manager
  VAR
    Filters_204A : Burkert.DO_UDFB;
    Filters_204B : Burkert.DO_UDFB;
    Filters_205A : Burkert.DO_UDFB;
    Filters_205B : Burkert.DO_UDFB;
    Stack_B : Burkert.DO_UDFB;
    Stack_G : Burkert.DO_UDFB;
    Stack_H : Burkert.DO_UDFB;
    Stack_R : Burkert.DO_UDFB;
    Filter_Skid : Burkert.DO_UDFB;
    TK201_PWR_1 : Burkert.DO_UDFB;
    TK201_PWR_2 : Burkert.DO_UDFB;
    TK201_PWR_3 : Burkert.DO_UDFB;
    Skid_201_PWR : Burkert.DO_UDFB;
    Skid_203_PWR : Burkert.DO_UDFB;
  END_VAR

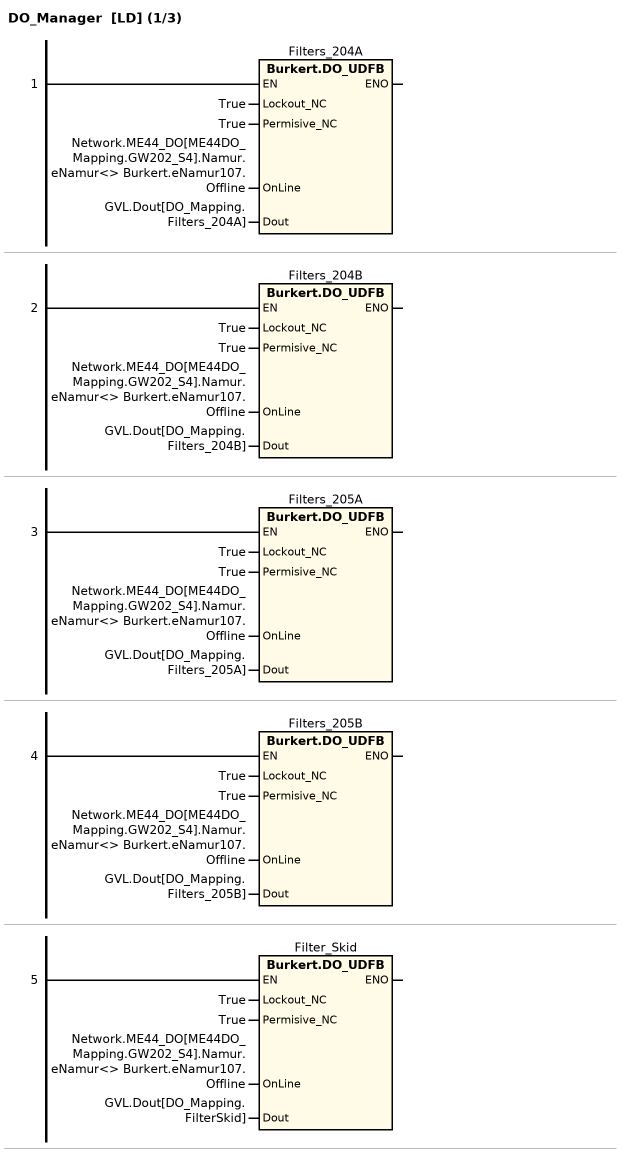
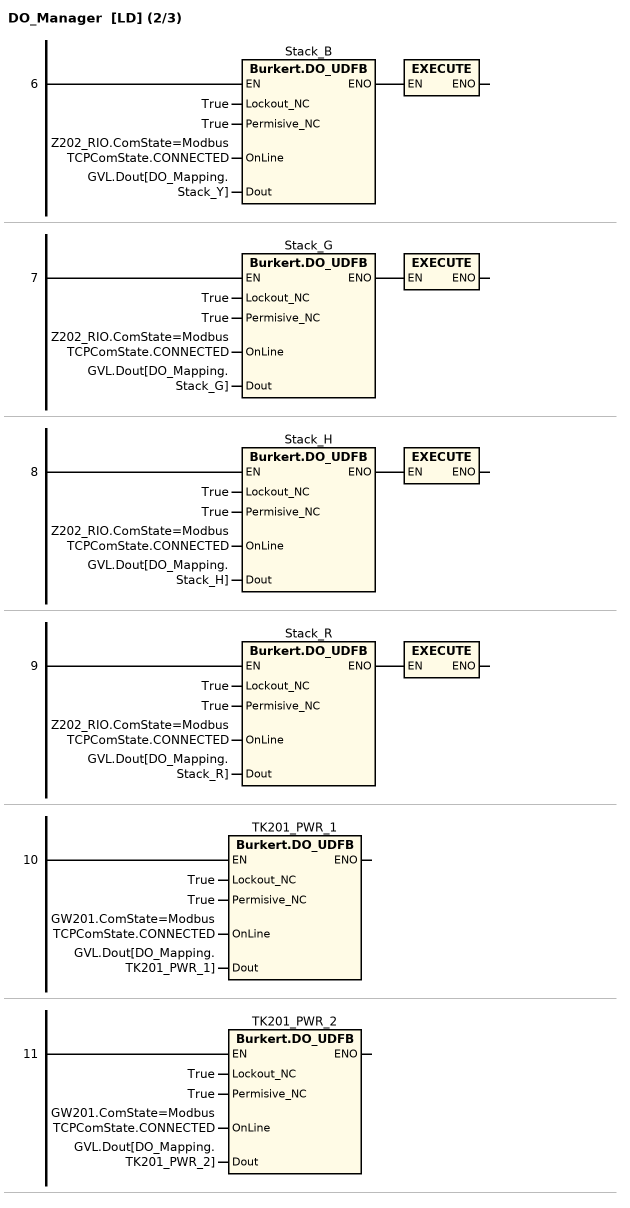
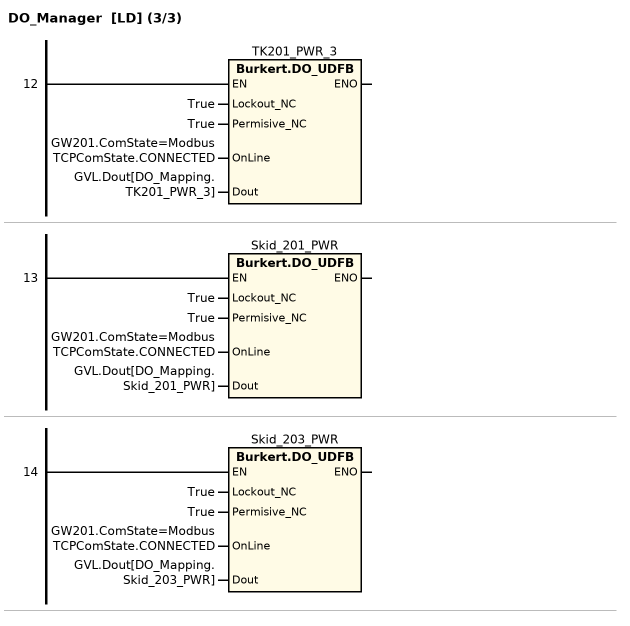
(* LD diagram, written out as Structured Text *)

Filters_204A(Lockout_NC := True, Permisive_NC := True, OnLine := Network.ME44_DO[ME44DO_Mapping.GW202_S4].Namur.eNamur<> Burkert.eNamur107.Offline, Dout := GVL.Dout[DO_Mapping.Filters_204A]);

Filters_204B(Lockout_NC := True, Permisive_NC := True, OnLine := Network.ME44_DO[ME44DO_Mapping.GW202_S4].Namur.eNamur<> Burkert.eNamur107.Offline, Dout := GVL.Dout[DO_Mapping.Filters_204B]);

Filters_205A(Lockout_NC := True, Permisive_NC := True, OnLine := Network.ME44_DO[ME44DO_Mapping.GW202_S4].Namur.eNamur<> Burkert.eNamur107.Offline, Dout := GVL.Dout[DO_Mapping.Filters_205A]);

Filters_205B(Lockout_NC := True, Permisive_NC := True, OnLine := Network.ME44_DO[ME44DO_Mapping.GW202_S4].Namur.eNamur<> Burkert.eNamur107.Offline, Dout := GVL.Dout[DO_Mapping.Filters_205B]);

Filter_Skid(Lockout_NC := True, Permisive_NC := True, OnLine := Network.ME44_DO[ME44DO_Mapping.GW202_S4].Namur.eNamur<> Burkert.eNamur107.Offline, Dout := GVL.Dout[DO_Mapping.FilterSkid]);


Stack_B(Lockout_NC := True, Permisive_NC := True, OnLine := Z202_RIO.ComState=ModbusTCPComState.CONNECTED, Dout := GVL.Dout[DO_Mapping.Stack_Y]);
IF Stack_B.ENO THEN
  Network.Z202_SIO_MB12CDR.Dout[2]:=GVL.Dout[DO_Mapping.Stack_Y].Q;
END_IF;

Stack_G(Lockout_NC := True, Permisive_NC := True, OnLine := Z202_RIO.ComState=ModbusTCPComState.CONNECTED, Dout := GVL.Dout[DO_Mapping.Stack_G]);
IF Stack_G.ENO THEN
  Network.Z202_SIO_MB12CDR.Dout[3]:=GVL.Dout[DO_Mapping.Stack_G].Q;
END_IF;

Stack_H(Lockout_NC := True, Permisive_NC := True, OnLine := Z202_RIO.ComState=ModbusTCPComState.CONNECTED, Dout := GVL.Dout[DO_Mapping.Stack_H]);
IF Stack_H.ENO THEN
  Network.Z202_SIO_MB12CDR.Dout[0]:=GVL.Dout[DO_Mapping.Stack_H].Q;
END_IF;

Stack_R(Lockout_NC := True, Permisive_NC := True, OnLine := Z202_RIO.ComState=ModbusTCPComState.CONNECTED, Dout := GVL.Dout[DO_Mapping.Stack_R]);
IF Stack_R.ENO THEN
  Network.Z202_SIO_MB12CDR.Dout[1]:=GVL.Dout[DO_Mapping.Stack_R].Q;
END_IF;

TK201_PWR_1(Lockout_NC := True, Permisive_NC := True, OnLine := GW201.ComState=ModbusTCPComState.CONNECTED, Dout := GVL.Dout[DO_Mapping.TK201_PWR_1]);

TK201_PWR_2(Lockout_NC := True, Permisive_NC := True, OnLine := GW201.ComState=ModbusTCPComState.CONNECTED, Dout := GVL.Dout[DO_Mapping.TK201_PWR_2]);

TK201_PWR_3(Lockout_NC := True, Permisive_NC := True, OnLine := GW201.ComState=ModbusTCPComState.CONNECTED, Dout := GVL.Dout[DO_Mapping.TK201_PWR_3]);

Skid_201_PWR(Lockout_NC := True, Permisive_NC := True, OnLine := GW201.ComState=ModbusTCPComState.CONNECTED, Dout := GVL.Dout[DO_Mapping.Skid_201_PWR]);

Skid_203_PWR(Lockout_NC := True, Permisive_NC := True, OnLine := GW201.ComState=ModbusTCPComState.CONNECTED, Dout := GVL.Dout[DO_Mapping.Skid_203_PWR]);
(* --- network --- *)
END_PROGRAM

PROGRAM Duplex_Manager
  VAR
    Z100_CTRL : Burkert.Duplex_VFD;
  END_VAR

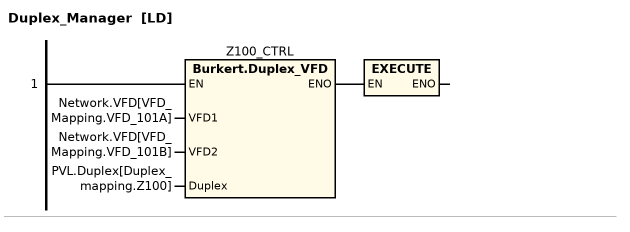
(* LD diagram, written out as Structured Text *)

Z100_CTRL(VFD1 := Network.VFD[VFD_Mapping.VFD_101A], VFD2 := Network.VFD[VFD_Mapping.VFD_101B], Duplex := PVL.Duplex[Duplex_mapping.Z100]);
IF Z100_CTRL.ENO THEN
  IF NOT(GVL.s3363[s3363_Mapping.ACV_101].Ready) AND (GVL.s3363[s3363_Mapping.ACV_102].Ready) AND 
  	(PVL.Duplex[Duplex_mapping.Z100].mode.emode =Burkert.eDuplex_Mode.Auto OR PVL.Duplex[Duplex_mapping.Z100].mode.emode =Burkert.eDuplex_Mode.Force_1) THEN
  	PVL.Duplex[Duplex_mapping.Z100].mode.emode:=Burkert.eDuplex_mode.Disabled;
  END_IF;
  
  IF (GVL.s3363[s3363_Mapping.ACV_101].Ready) AND NOT(GVL.s3363[s3363_Mapping.ACV_102].Ready) AND	
  	(PVL.Duplex[Duplex_mapping.Z100].mode.emode =Burkert.eDuplex_Mode.Auto OR PVL.Duplex[Duplex_mapping.Z100].mode.emode =Burkert.eDuplex_Mode.Force_2) THEN
  	PVL.Duplex[Duplex_mapping.Z100].mode.emode:=Burkert.eDuplex_mode.Disabled;
  END_IF;
  
  IF NOT(GVL.s3363[s3363_Mapping.ACV_101].Ready) AND NOT(GVL.s3363[s3363_Mapping.ACV_102].Ready) THEN
  	PVL.Duplex[Duplex_mapping.Z100].mode.emode:=Burkert.eDuplex_mode.Disabled;
  END_IF;
END_IF;
END_PROGRAM

PROGRAM Level_2_CTRL

            PID_Manager();
Duplex_Manager();
Stack_Light_CTRL();


          
END_PROGRAM

PROGRAM Stack_Light_CTRL
  VAR
    Stack_Lights_4Way_0 : Burkert.Stack_Lights_4Way;
    Warning : BOOL;
    Alarm : BOOL;
    Index : INT;
    CLK_Prg : Burkert.Burkert_OSCAT_BASIC.CLK_PRG;
  END_VAR
  VAR  (* added by the conversion: wires and edge detectors of the diagram *)
    _AND11_OUT : BOOL;
    _Warnings36_OUT : ANY;
    _Warnings36_ENO : BOOL;
  END_VAR

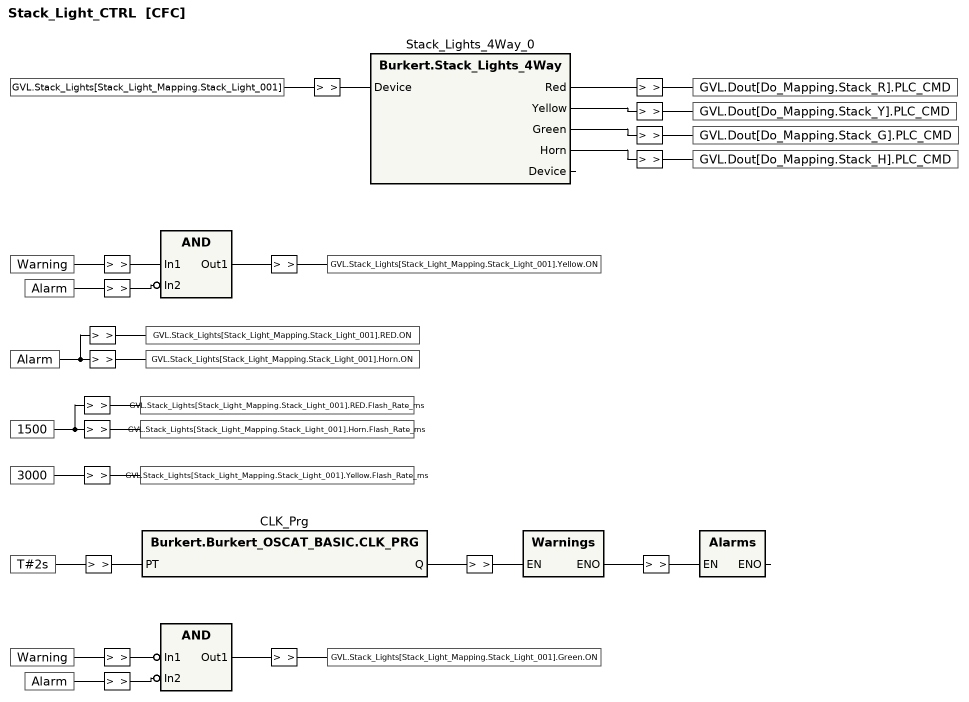
(* CFC diagram, written out as Structured Text *)
GVL.Dout[Do_Mapping.Stack_G].PLC_CMD := Stack_Lights_4Way_0.Green;
GVL.Dout[Do_Mapping.Stack_H].PLC_CMD := Stack_Lights_4Way_0.Horn;
GVL.Dout[Do_Mapping.Stack_Y].PLC_CMD := Stack_Lights_4Way_0.Yellow;
GVL.Stack_Lights[Stack_Light_Mapping.Stack_Light_001].Yellow.ON := _AND11_OUT;
_AND11_OUT := Warning AND NOT Alarm;
GVL.Stack_Lights[Stack_Light_Mapping.Stack_Light_001].RED.ON := Alarm;
GVL.Stack_Lights[Stack_Light_Mapping.Stack_Light_001].RED.Flash_Rate_ms := 1500;
Stack_Lights_4Way_0(Device := GVL.Stack_Lights[Stack_Light_Mapping.Stack_Light_001]);
GVL.Stack_Lights[Stack_Light_Mapping.Stack_Light_001].Yellow.Flash_Rate_ms := 3000;
GVL.Stack_Lights[Stack_Light_Mapping.Stack_Light_001].Horn.ON := Alarm;
GVL.Stack_Lights[Stack_Light_Mapping.Stack_Light_001].Horn.Flash_Rate_ms := 1500;
GVL.Dout[Do_Mapping.Stack_R].PLC_CMD := Stack_Lights_4Way_0.Red;
CLK_Prg(PT := T#2s);
IF _Warnings36_OUT THEN Alarms(); END_IF;
_Warnings36_OUT := Warnings(EN := CLK_Prg.Q, ENO => _Warnings36_ENO);
GVL.Stack_Lights[Stack_Light_Mapping.Stack_Light_001].Green.ON := NOT Warning AND NOT Alarm;

ACTION Warnings:
                Warning:=FALSE;

FOR Index:=0 TO AIT_Mapping.AIT_End-1 BY 1 DO
	IF PVl.AIT[index].Status.eStatus=Burkert.eSensor_Status.High_Warning OR PVl.AIT[index].Status.eStatus=Burkert.eSensor_Status.Low_Warning THEN Warning:=TRUE; END_IF;
END_FOR;

FOR Index:=0 TO s8312_Mapping.S8312_End-1 BY 1 DO
	IF PVl.s8312[Index].Status.eStatus=Burkert.eSensor_Status.High_Warning OR PVl.s8312[index].Status.eStatus=Burkert.eSensor_Status.Low_Warning THEN Warning:=TRUE; END_IF;
END_FOR;

FOR Index:=0 TO s8098_Mapping.S8098_End-1 BY 1 DO
	IF PVl.s8098[Index].PDO.VolumeFlow.Status.eStatus=Burkert.eSensor_Status.High_Warning OR PVl.s8098[index].PDO.VolumeFlow.Status.eStatus =Burkert.eSensor_Status.Low_Warning THEN Warning:=TRUE; END_IF;
END_FOR;


              
END_ACTION

ACTION Alarms:
                Alarm:=FALSE;

FOR Index:=0 TO AIT_Mapping.AIT_End-1 BY 1 DO
	IF PVl.AIT[index].Status.eStatus=Burkert.eSensor_Status.Low_Low_Alarm OR PVl.AIT[index].Status.eStatus=Burkert.eSensor_Status.HiHi_Alarm THEN Alarm:=TRUE; END_IF;
END_FOR;

FOR Index:=0 TO s8312_Mapping.S8312_End-1 BY 1 DO
	IF PVl.s8312[Index].Status.eStatus=Burkert.eSensor_Status.Low_Low_Alarm OR PVl.s8312[index].Status.eStatus=Burkert.eSensor_Status.HiHi_Alarm THEN Alarm:=TRUE; END_IF;
END_FOR;

FOR Index:=0 TO s8098_Mapping.S8098_End-1 BY 1 DO
	IF PVl.s8098[Index].PDO.VolumeFlow.Status.eStatus=Burkert.eSensor_Status.Low_Low_Alarm OR PVl.s8098[index].PDO.VolumeFlow.Status.eStatus =Burkert.eSensor_Status.HiHi_Alarm THEN Alarm:=TRUE; END_IF;
END_FOR;


              
END_ACTION
END_PROGRAM

PROGRAM Z202_Manager
  VAR
    Local_Status : eZ202_Status;
    tStatus : eZ202_Status;  (* P203_Local_Status:eZ202_Status; *)
    Local_Task : eZ202_Task;
    tAlarm : Burkert.Alarm_Window;  (* P203_Local_Task:eZ202_Task; *)
    Task_Ton : Ton;
    Valve_Ton : Ton;
    SubIndex : UINT;
    lcl_Valve_Matrix : WORD;
    FT202_Ave : REAL;
    FT202_Gav : REAL;
    FT202_Hav : REAL;
    FT202_Ave_Index : INT;
    FT202_Array_Size : UINT;
    FT203_Ave : REAL;
    FT203_Gav : REAL;
    FT203_Hav : REAL;
    FT203_Ave_Index : INT;
    FT203_Array_Size : UINT;
    Level_Ton : Ton;
    Min_Pump_Speed : REAL := 10;
    RS_ACV_203 : RS;
    RAMP_REAL_0 : Burkert.RAMP_REAL;
    RAMP_REAL_1 : Burkert.RAMP_REAL;
  END_VAR
  VAR  (* added by the conversion: wires and edge detectors of the diagram *)
    _OR123_OUT : BOOL;
    _AND161_OUT : BOOL;
    _AND185_OUT : BOOL;
    _OR14_OUT : BOOL;
    _OR24_OUT : BOOL;
    _OR48_OUT : BOOL;
    _OR66_OUT : BOOL;
    _OR241_OUT : BOOL;
    _OR187_OUT : BOOL;
    _OR207_OUT : BOOL;
    _SEL4_OUT : ANY;
    _AND253_OUT : BOOL;
    _OR255_OUT : BOOL;
    _OR271_OUT : BOOL;
    _OR164_OUT : BOOL;
    _OR2_OUT : BOOL;
    _OR29_OUT : BOOL;
    _AND44_OUT : BOOL;
    _GT2_OUT : BOOL;
    _OR18_OUT : BOOL;
    _OR35_OUT : BOOL;
    _SEL80_OUT : ANY;
    _MAX122_OUT : ANY;
    _SEL84_OUT : ANY;
    _OR6_OUT : BOOL;
    _SEL14_OUT : ANY;
    _SEL4_OUT_2 : ANY;
    _AND16_OUT : BOOL;
    _SEL30_OUT : ANY;
  END_VAR

            Aux();
Alarms();


//Test_Conflict();

PVL.Z202_Config.StrMode:=Burkert.Burkert_OSCAT_BASIC.REPLACE_ALL(str:=TO_STRING(PVL.Z202_Config.Mode.eMode) , src:='_' , rep:=' ' );
PVL.Z202_Config.StrStatus:=Burkert.Burkert_OSCAT_BASIC.REPLACE_ALL(str:=TO_STRING(PVL.Z202_Config.Status.eStatus) , src:='_' , rep:=' ' );
PVL.Z202_Config.Mode.eMode:=Burkert.eHOA_Modes.Manual;
PVl.Z202_Config.StrTask:=Burkert.Burkert_OSCAT_BASIC.REPLACE_ALL(str:=TO_STRING(PVL.Z202_Config.Task.eTask) , src:='_' , rep:=' ' );
//PVL.Z202_Config.P203_StrStatus:=Burkert.Burkert_OSCAT_BASIC.REPLACE_ALL(str:=TO_STRING(PVL.Z202_Config.P203_Status.eStatus) , src:='_' , rep:=' ' );
//PVl.Z202_Config.P203_StrTask:=Burkert.Burkert_OSCAT_BASIC.REPLACE_ALL(str:=TO_STRING(PVL.Z202_Config.P203_Task.eTask) , src:='_' , rep:=' ' );




CASE PVL.Z202_Config.Mode.eMode OF
	Burkert.eHOA_Modes.Off:
		PVL.Z202_Config.Task.eTask:=eZ202_task.Off;
		//PVL.Z202_Config.P203_Task.eTask:=eZ202_task.Off;
	Burkert.eHOA_Modes.Auto:	Mode_Auto();
	//Burkert.eHOA_Modes.Manual:
END_CASE;

CASE pvl.Z202_Config.Task.eTask OF
	eZ202_Task.Off:		Task_Off();
	eZ202_Task.TK201_Level_Return_P202:		TK201_Level_Return_P202();
	eZ202_task.Rate_Return_P202:			Rate_Return_P202();
	eZ202_Task.Filter_Level_P202:			Filter_Level_P202();
	eZ202_Task.Filter_Flow_P202:			Filter_Flow_P202();
	eZ202_Task.Recovery_Rate_P202:			Recovery_Rate_P202();
	eZ202_Task.Recovery_Speed_P202:			Recovery_Speed_P202();
	eZ202_Task.Drain_P202:				Drain_P202();
	
END_CASE

CASE pvl.Z202_Config.Task.eTask OF
	//eZ202_Task.Off:		Task_Off();
	eZ202_Task.TK201_Level_Return_P203:		TK201_Level_Return_P203();
	eZ202_task.EP101_Level_Return_P203:		EP101_Level_Return_P203();
	eZ202_Task.Filter_Level_P203:			Filter_Level_P203();
	eZ202_Task.Filter_Flow_P203:			Filter_Flow_P203();
	eZ202_task.Rate_Return_P203:			Rate_Return_P203();
	eZ202_Task.Recovery_Speed_P203:			Recovery_Speed_P203();
	eZ202_Task.Recovery_Rate_P203:			Recovery_Rate_P203();
	eZ202_Task.Drain_P203:					Drain_P203();
END_CASE

CASE pvl.Z202_Config.Task.eTask OF
	eZ202_task.Filter_Level_P202_Recovery_Speed_P203:	Filter_Level_P202_Recovery_Speed_P203();
	eZ202_task.Filter_Flow_P202_Recovery_Speed_P203:	Filter_Flow_P202_Recovery_Speed_P203();
	eZ202_task.Filter_Level_P202_Recovery_Flow_P203:	Filter_Level_P202_Recovery_Flow_P203();
	eZ202_task.Filter_Flow_P202_Recovery_Flow_P203:		Filter_Flow_P202_Recovery_Flow_P203();
	
END_CASE



PID_ctrl();
ACV_ctrl();
VFD_ctrl();
          

ACTION Test_P203_Conflict:
                (*
CASE PVL.Z202_Config.P203_Task.eTask OF
	eZ202_Task.EP101_Level_Return_P203:
		CASE PVl.Z202_Config.P202_Task.eTask OF
			eZ202_Task.EP101_Level_Return_P202:PVL.Z202_Config.P202_Task.eTask:=eZ202_Task.Off;
			eZ202_Task.Filter_Flow_P202:
			eZ202_Task.Filter_Level_P202:
			eZ202_Task.Rate_Return_P202:PVL.Z202_Config.P202_Task.eTask:=eZ202_Task.Off;
			eZ202_Task.Recovery_Rate_P202:PVL.Z202_Config.P202_Task.eTask:=eZ202_Task.Off;
			eZ202_Task.Recovery_Speed_P202:PVL.Z202_Config.P202_Task.eTask:=eZ202_Task.Off;
			eZ202_Task.TK201_Level_Return_P202:PVL.Z202_Config.P202_Task.eTask:=eZ202_Task.Off;
		END_CASE
	eZ202_Task.Filter_Flow_P203:
		CASE PVl.Z202_Config.P202_Task.eTask OF
			eZ202_Task.EP101_Level_Return_P202:
			eZ202_Task.Filter_Flow_P202:PVL.Z202_Config.P202_Task.eTask:=eZ202_Task.Off;
			eZ202_Task.Filter_Level_P202:PVL.Z202_Config.P202_Task.eTask:=eZ202_Task.Off;
			eZ202_Task.Rate_Return_P202:
			eZ202_Task.Recovery_Rate_P202:
			eZ202_Task.Recovery_Speed_P202:
			eZ202_Task.TK201_Level_Return_P202:
		END_CASE
	eZ202_Task.Filter_Level_P203:
		CASE PVl.Z202_Config.P202_Task.eTask OF
			eZ202_Task.EP101_Level_Return_P202:
			eZ202_Task.Filter_Flow_P202:PVL.Z202_Config.P202_Task.eTask:=eZ202_Task.Off;
			eZ202_Task.Filter_Level_P202:PVL.Z202_Config.P202_Task.eTask:=eZ202_Task.Off;
			eZ202_Task.Rate_Return_P202:
			eZ202_Task.Recovery_Rate_P202:
			eZ202_Task.Recovery_Speed_P202:
			eZ202_Task.TK201_Level_Return_P202:
		END_CASE
	eZ202_Task.Rate_Return_P203:
		CASE PVl.Z202_Config.P202_Task.eTask OF
			eZ202_Task.EP101_Level_Return_P202:PVL.Z202_Config.P202_Task.eTask:=eZ202_Task.Off;
			eZ202_Task.Filter_Flow_P202:
			eZ202_Task.Filter_Level_P202:
			eZ202_Task.Rate_Return_P202:PVL.Z202_Config.P202_Task.eTask:=eZ202_Task.Off;
			eZ202_Task.Recovery_Rate_P202:PVL.Z202_Config.P202_Task.eTask:=eZ202_Task.Off;
			eZ202_Task.Recovery_Speed_P202:PVL.Z202_Config.P202_Task.eTask:=eZ202_Task.Off;
			eZ202_Task.TK201_Level_Return_P202:PVL.Z202_Config.P202_Task.eTask:=eZ202_Task.Off;
		END_CASE
	eZ202_Task.Recovery_Rate_P203:
		CASE PVl.Z202_Config.P202_Task.eTask OF
			eZ202_Task.EP101_Level_Return_P202:PVL.Z202_Config.P202_Task.eTask:=eZ202_Task.Off;
			eZ202_Task.Filter_Flow_P202:
			eZ202_Task.Filter_Level_P202:
			eZ202_Task.Rate_Return_P202:PVL.Z202_Config.P202_Task.eTask:=eZ202_Task.Off;
			eZ202_Task.Recovery_Rate_P202:PVL.Z202_Config.P202_Task.eTask:=eZ202_Task.Off;
			eZ202_Task.Recovery_Speed_P202:PVL.Z202_Config.P202_Task.eTask:=eZ202_Task.Off;
			eZ202_Task.TK201_Level_Return_P202:PVL.Z202_Config.P202_Task.eTask:=eZ202_Task.Off;
		END_CASE
	eZ202_Task.Recovery_Speed_P203:
		CASE PVl.Z202_Config.P202_Task.eTask OF
			eZ202_Task.EP101_Level_Return_P202:PVL.Z202_Config.P202_Task.eTask:=eZ202_Task.Off;
			eZ202_Task.Filter_Flow_P202:
			eZ202_Task.Filter_Level_P202:
			eZ202_Task.Rate_Return_P202:PVL.Z202_Config.P202_Task.eTask:=eZ202_Task.Off;
			eZ202_Task.Recovery_Rate_P202:PVL.Z202_Config.P202_Task.eTask:=eZ202_Task.Off;
			eZ202_Task.Recovery_Speed_P202:PVL.Z202_Config.P202_Task.eTask:=eZ202_Task.Off;
			eZ202_Task.TK201_Level_Return_P202:PVL.Z202_Config.P202_Task.eTask:=eZ202_Task.Off;
		END_CASE
	eZ202_Task.TK201_Level_Return_P203:
		CASE PVl.Z202_Config.P202_Task.eTask OF
			eZ202_Task.EP101_Level_Return_P202:PVL.Z202_Config.P202_Task.eTask:=eZ202_Task.Off;
			eZ202_Task.Filter_Flow_P202:
			eZ202_Task.Filter_Level_P202:
			eZ202_Task.Rate_Return_P202:PVL.Z202_Config.P202_Task.eTask:=eZ202_Task.Off;
			eZ202_Task.Recovery_Rate_P202:PVL.Z202_Config.P202_Task.eTask:=eZ202_Task.Off;
			eZ202_Task.Recovery_Speed_P202:PVL.Z202_Config.P202_Task.eTask:=eZ202_Task.Off;
			eZ202_Task.TK201_Level_Return_P202:PVL.Z202_Config.P202_Task.eTask:=eZ202_Task.Off;
		END_CASE
	
END_CASE
*)
              
END_ACTION

ACTION ACV_ctrl:
